LIN {X 0,Y 240.149,Z 360.494,A -85,B 0,C 180,E1 -19958.542,E2 -19958.542} C_VEL
LIN {X 0,Y 236.743,Z 363.17,A -85,B 0,C 180,E1 -19960.941,E2 -19960.941} C_VEL
LIN {X 0,Y 232.958,Z 365.456,A -85,B 0,C 180,E1 -19964.245,E2 -19964.245} C_VEL
LIN {X 0,Y 230.136,Z 366.365,A -85,B 0,C 180,E1 -19967.657,E2 -19967.657} C_VEL
LIN {X 0,Y 228.663,Z 366.29,A -85,B 0,C 180,E1 -19969.595,E2 -19969.595} C_VEL
LIN {X 0,Y 227.257,Z 365.084,A -85,B 0,C 180,E1 -19972.894,E2 -19972.894} C_VEL
LIN {X 0,Y 226.376,Z 362.416,A -85,B 0,C 180,E1 -19976.44,E2 -19976.44} C_VEL
LIN {X 0,Y 225.981,Z 359.392,A -85,B 0,C 180,E1 -19979.109,E2 -19979.109} C_VEL
LIN {X 0,Y 225.959,Z 355.435,A -85,B 0,C 180,E1 -19981.782,E2 -19981.782} C_VEL
LIN {X 0,Y 226.033,Z 350.41,A -85,B 0,C 180,E1 -19984.458,E2 -19984.458} C_VEL
LIN {X 0,Y 226.423,Z 343.052,A -85,B 0,C 180,E1 -19987.58,E2 -19987.58} C_VEL
LIN {X 0,Y 227.138,Z 333.719,A -85,B 0,C 180,E1 -19990.699,E2 -19990.699} C_VEL
LIN {X 0,Y 228.026,Z 323.757,A -85,B 0,C 180,E1 -19993.365,E2 -19993.365} C_VEL
LIN {X 0,Y 229.272,Z 312.636,A -85,B 0,C 180,E1 -19995.786,E2 -19995.786} C_VEL
LIN {X 0,Y 230.346,Z 301.437,A -85,B 0,C 180,E1 -19997.765,E2 -19997.765} C_VEL
LIN {X 0,Y 231.551,Z 289.361,A -85,B 0,C 180,E1 -19999.504,E2 -19999.504} C_VEL
LIN {X 0,Y 231.875,Z 284.182,A -85,B 0,C 180,E1 -20000.139,E2 -20000.139} C_VEL
LIN {X 0,Y 229.783,Z 269.787,A -85,B 0,C 180,E1 -20001.668,E2 -20001.668} C_VEL
LIN {X 0,Y 228.207,Z 255.116,A -85,B 0,C 180,E1 -20002.85,E2 -20002.85} C_VEL
LIN {X 0,Y 228.789,Z 246.393,A -85,B 0,C 180,E1 -20007.437,E2 -20007.437} C_VEL
LIN {X 0,Y 229.412,Z 238.95,A -85,B 0,C 180,E1 -20011.386,E2 -20011.386} C_VEL
LIN {X 0,Y 230.076,Z 231.264,A -85,B 0,C 180,E1 -20015.478,E2 -20015.478} C_VEL
LIN {X 0,Y 229.952,Z 226.244,A -85,B 0,C 180,E1 -20018.23,E2 -20018.23} C_VEL
LIN {X 0,Y 228.576,Z 218.639,A -85,B 0,C 180,E1 -20022.566,E2 -20022.566} C_VEL
LIN {X 0,Y 227.886,Z 215.096,A -85,B 0,C 180,E1 -20024.661,E2 -20024.661} C_VEL
LIN {X 0,Y 227.869,Z 215.294,A -85,B 0,C 180,E1 -20027.269,E2 -20027.269} C_VEL
LIN {X 0,Y 228.539,Z 218.744,A -85,B 0,C 180,E1 -20032.043,E2 -20032.043} C_VEL
LIN {X 0,Y 229.088,Z 222.169,A -85,B 0,C 180,E1 -20036.479,E2 -20036.479} C_VEL
LIN {X 0,Y 229.253,Z 224.421,A -85,B 0,C 180,E1 -20039.135,E2 -20039.135} C_VEL
LIN {X 0,Y 229.175,Z 227.751,A -85,B 0,C 180,E1 -20042.789,E2 -20042.789} C_VEL
LIN {X 0,Y 228.957,Z 231.942,A -85,B 0,C 180,E1 -20047.054,E2 -20047.054} C_VEL
LIN {X 0,Y 232.523,Z 242.538,A -85,B 0,C 180,E1 -20048.242,E2 -20048.242} C_VEL
LIN {X 0,Y 234.853,Z 251.139,A -85,B 0,C 180,E1 -20049.409,E2 -20049.409} C_VEL
LIN {X 0,Y 236.685,Z 260.451,A -85,B 0,C 180,E1 -20050.934,E2 -20050.934} C_VEL
LIN {X 0,Y 237.154,Z 263.439,A -85,B 0,C 180,E1 -20051.499,E2 -20051.499} C_VEL
LIN {X 0,Y 236.153,Z 271.037,A -85,B 0,C 180,E1 -20052.907,E2 -20052.907} C_VEL
LIN {X 0,Y 234.935,Z 277.492,A -85,B 0,C 180,E1 -20054.379,E2 -20054.379} C_VEL
LIN {X 0,Y 233.482,Z 283.544,A -85,B 0,C 180,E1 -20056.064,E2 -20056.064} C_VEL
LIN {X 0,Y 232.2,Z 288.356,A -85,B 0,C 180,E1 -20057.766,E2 -20057.766} C_VEL
LIN {X 0,Y 231.114,Z 292.243,A -85,B 0,C 180,E1 -20059.485,E2 -20059.485} C_VEL
LIN {X 0,Y 230.298,Z 296.589,A -85,B 0,C 180,E1 -20062.105,E2 -20062.105} C_VEL
LIN {X 0,Y 229.216,Z 299.558,A -85,B 0,C 180,E1 -20064.72,E2 -20064.72} C_VEL
LIN {X 0,Y 228.932,Z 300.802,A -85,B 0,C 180,E1 -20066.478,E2 -20066.478} C_VEL
LIN {X 0,Y 228.662,Z 301.565,A -85,B 0,C 180,E1 -20068.236,E2 -20068.236} C_VEL
LIN {X 0,Y 228.557,Z 301.836,A -85,B 0,C 180,E1 -20069.998,E2 -20069.998} C_VEL
LIN {X 0,Y 228.661,Z 301.599,A -85,B 0,C 180,E1 -20071.759,E2 -20071.759} C_VEL
LIN {X 0,Y 228.93,Z 300.884,A -85,B 0,C 180,E1 -20073.518,E2 -20073.518} C_VEL
LIN {X 0,Y 229.213,Z 299.688,A -85,B 0,C 180,E1 -20075.275,E2 -20075.275} C_VEL
LIN {X 0,Y 230.285,Z 296.77,A -85,B 0,C 180,E1 -20077.891,E2 -20077.891} C_VEL
LIN {X 0,Y 231.073,Z 292.516,A -85,B 0,C 180,E1 -20080.512,E2 -20080.512} C_VEL
LIN {X 0,Y 231.808,Z 290.679,A -85,B 0,C 180,E1 -20081.363,E2 -20081.363} C_VEL
LIN {X 0,Y 232.744,Z 286.458,A -85,B 0,C 180,E1 -20083.087,E2 -20083.087} C_VEL
LIN {X 0,Y 234.536,Z 279.688,A -85,B 0,C 180,E1 -20085.198,E2 -20085.198} C_VEL
LIN {X 0,Y 235.91,Z 272.696,A -85,B 0,C 180,E1 -20086.883,E2 -20086.883} C_VEL
LIN {X 0,Y 236.953,Z 265.692,A -85,B 0,C 180,E1 -20088.245,E2 -20088.245} C_VEL
LIN {X 0,Y 237.125,Z 263.241,A -85,B 0,C 180,E1 -20088.68,E2 -20088.68} C_VEL
LIN {X 0,Y 235.737,Z 254.873,A -85,B 0,C 180,E1 -20090.151,E2 -20090.151} C_VEL
LIN {X 0,Y 233.638,Z 246.157,A -85,B 0,C 180,E1 -20091.422,E2 -20091.422} C_VEL
LIN {X 0,Y 230.323,Z 235.832,A -85,B 0,C 180,E1 -20092.688,E2 -20092.688} C_VEL
LIN {X 0,Y 228.951,Z 231.943,A -85,B 0,C 180,E1 -20093.098,E2 -20093.098} C_VEL
LIN {X 0,Y 229.195,Z 227.77,A -85,B 0,C 180,E1 -20097.382,E2 -20097.382} C_VEL
LIN {X 0,Y 229.217,Z 224.148,A -85,B 0,C 180,E1 -20101.412,E2 -20101.412} C_VEL
LIN {X 0,Y 229.06,Z 221.908,A -85,B 0,C 180,E1 -20104.064,E2 -20104.064} C_VEL
LIN {X 0,Y 228.562,Z 218.862,A -85,B 0,C 180,E1 -20107.947,E2 -20107.947} C_VEL
LIN {X 0,Y 227.893,Z 215.434,A -85,B 0,C 180,E1 -20112.72,E2 -20112.72} C_VEL
LIN {X 0,Y 227.863,Z 215.098,A -85,B 0,C 180,E1 -20113.941,E2 -20113.941} C_VEL
LIN {X 0,Y 227.859,Z 215.104,A -85,B 0,C 180,E1 -20117.748,E2 -20117.748} C_VEL
LIN {X 0,Y 227.859,Z 215.097,A -85,B 0,C 180,E1 -20121.912,E2 -20121.912} C_VEL
LIN {X 0,Y 227.877,Z 215.09,A -85,B 0,C 180,E1 -20126.373,E2 -20126.373} C_VEL
LIN {X 0,Y 227.911,Z 215.084,A -85,B 0,C 180,E1 -20130.436,E2 -20130.436} C_VEL
LIN {X 0,Y 227.92,Z 215.082,A -85,B 0,C 180,E1 -20134.425,E2 -20134.425} C_VEL
LIN {X 0,Y 227.953,Z 215.086,A -85,B 0,C 180,E1 -20138.286,E2 -20138.286} C_VEL
LIN {X 0,Y 228.025,Z 215.081,A -85,B 0,C 180,E1 -20142.825,E2 -20142.825} C_VEL
LIN {X 0,Y 228.063,Z 215.078,A -85,B 0,C 180,E1 -20147.543,E2 -20147.543} C_VEL
LIN {X 0,Y 228.257,Z 215.041,A -85,B 0,C 180,E1 -20151.144,E2 -20151.144} C_VEL
LIN {X 0,Y 228.329,Z 215.043,A -85,B 0,C 180,E1 -20152.928,E2 -20152.928} C_VEL
LIN {X 0,Y 228.544,Z 215.014,A -85,B 0,C 180,E1 -20158.238,E2 -20158.238} C_VEL
LIN {X 0,Y 228.543,Z 215.013,A -85,B 0,C 180,E1 -20161.762,E2 -20161.762} C_VEL
LIN {X 0,Y 228.344,Z 215.042,A -85,B 0,C 180,E1 -20167.072,E2 -20167.072} C_VEL
LIN {X 0,Y 228.148,Z 215.062,A -85,B 0,C 180,E1 -20170.651,E2 -20170.651} C_VEL
LIN {X 0,Y 228.031,Z 215.072,A -85,B 0,C 180,E1 -20174.274,E2 -20174.274} C_VEL
LIN {X 0,Y 227.919,Z 215.085,A -85,B 0,C 180,E1 -20177.96,E2 -20177.96} C_VEL
LIN {X 0,Y 227.878,Z 215.101,A -85,B 0,C 180,E1 -20182.304,E2 -20182.304} C_VEL
LIN {X 0,Y 227.893,Z 215.101,A -85,B 0,C 180,E1 -20186.584,E2 -20186.584} C_VEL
LIN {X 0,Y 227.88,Z 215.289,A -85,B 0,C 180,E1 -20188.809,E2 -20188.809} C_VEL
LIN {X 0,Y 229.216,Z 220.372,A -85,B 0,C 180,E1 -20193.497,E2 -20193.497} C_VEL
LIN {X 0,Y 230.426,Z 225.395,A -85,B 0,C 180,E1 -20197.59,E2 -20197.59} C_VEL
LIN {X 0,Y 231.746,Z 231.311,A -85,B 0,C 180,E1 -20201.85,E2 -20201.85} C_VEL
LIN {X 0,Y 233.255,Z 238.212,A -85,B 0,C 180,E1 -20206.313,E2 -20206.313} C_VEL
LIN {X 0,Y 234.535,Z 244.072,A -85,B 0,C 180,E1 -20209.828,E2 -20209.828} C_VEL
LIN {X 0,Y 235.471,Z 248.71,A -85,B 0,C 180,E1 -20212.45,E2 -20212.45} C_VEL
LIN {X 0,Y 235.38,Z 250.389,A -85,B 0,C 180,E1 -20213.311,E2 -20213.311} C_VEL
LIN {X 0,Y 233.997,Z 253.09,A -85,B 0,C 180,E1 -20214.552,E2 -20214.552} C_VEL
LIN {X 0,Y 231.754,Z 255.824,A -85,B 0,C 180,E1 -20215.736,E2 -20215.736} C_VEL
LIN {X 0,Y 227.007,Z 261.454,A -85,B 0,C 180,E1 -20218.199,E2 -20218.199} C_VEL
LIN {X 0,Y 226.091,Z 263.295,A -85,B 0,C 180,E1 -20219.09,E2 -20219.09} C_VEL
LIN {X 0,Y 224.786,Z 267.3,A -85,B 0,C 180,E1 -20221.096,E2 -20221.096} C_VEL
LIN {X 0,Y 225.919,Z 279.544,A -85,B 0,C 180,E1 -20222.011,E2 -20222.011} C_VEL
LIN {X 0,Y 226.392,Z 291.772,A -85,B 0,C 180,E1 -20223.251,E2 -20223.251} C_VEL
LIN {X 0,Y 226.184,Z 302.278,A -85,B 0,C 180,E1 -20224.585,E2 -20224.585} C_VEL
LIN {X 0,Y 225.585,Z 313.26,A -85,B 0,C 180,E1 -20226.355,E2 -20226.355} C_VEL
LIN {X 0,Y 225.14,Z 321.657,A -85,B 0,C 180,E1 -20228.004,E2 -20228.004} C_VEL
LIN {X 0,Y 224.202,Z 327.791,A -85,B 0,C 180,E1 -20229.353,E2 -20229.353} C_VEL
LIN {X 0,Y 222.571,Z 336.194,A -85,B 0,C 180,E1 -20231.596,E2 -20231.596} C_VEL
LIN {X 0,Y 221.338,Z 343.23,A -85,B 0,C 180,E1 -20233.872,E2 -20233.872} C_VEL
LIN {X 0,Y 220.649,Z 348.998,A -85,B 0,C 180,E1 -20236.182,E2 -20236.182} C_VEL
LIN {X 0,Y 220.308,Z 352.862,A -85,B 0,C 180,E1 -20238.035,E2 -20238.035} C_VEL
LIN {X 0,Y 219.852,Z 361.618,A -85,B 0,C 180,E1 -20240.805,E2 -20240.805} C_VEL
LIN {X 0,Y 219.728,Z 369.279,A -85,B 0,C 180,E1 -20243.851,E2 -20243.851} C_VEL
LIN {X 0,Y 219.716,Z 374.223,A -85,B 0,C 180,E1 -20246.334,E2 -20246.334} C_VEL
LIN {X 0,Y 219.799,Z 378.548,A -85,B 0,C 180,E1 -20249.086,E2 -20249.086} C_VEL
LIN {X 0,Y 219.482,Z 381.661,A -85,B 0,C 180,E1 -20251.837,E2 -20251.837} C_VEL
LIN {X 0,Y 218.975,Z 384.309,A -85,B 0,C 180,E1 -20255.528,E2 -20255.528} C_VEL
LIN {X 0,Y 219.193,Z 385.464,A -85,B 0,C 180,E1 -20259.228,E2 -20259.228} C_VEL
LIN {X 0,Y 220.33,Z 385.234,A -85,B 0,C 180,E1 -20262.904,E2 -20262.904} C_VEL
LIN {X 0,Y 222.524,Z 383.673,A -85,B 0,C 180,E1 -20266.516,E2 -20266.516} C_VEL
LIN {X 0,Y 225.922,Z 380.789,A -85,B 0,C 180,E1 -20270.012,E2 -20270.012} C_VEL
LIN {X 0,Y 230.072,Z 376.537,A -85,B 0,C 180,E1 -20273.4,E2 -20273.4} C_VEL
LIN {X 0,Y 234.016,Z 372.441,A -85,B 0,C 180,E1 -20275.817,E2 -20275.817} C_VEL
LIN {X 0,Y 240.311,Z 365.58,A -85,B 0,C 180,E1 -20278.854,E2 -20278.854} C_VEL
LIN {X 0,Y 246.571,Z 358.222,A -85,B 0,C 180,E1 -20281.346,E2 -20281.346} C_VEL
LIN {X 0,Y 253.528,Z 349.34,A -85,B 0,C 180,E1 -20283.673,E2 -20283.673} C_VEL
LIN {X 0,Y 259.702,Z 340.339,A -85,B 0,C 180,E1 -20285.677,E2 -20285.677} C_VEL
LIN {X 0,Y 264.058,Z 332.941,A -85,B 0,C 180,E1 -20287.267,E2 -20287.267} C_VEL
LIN {X 0,Y 268.671,Z 323.71,A -85,B 0,C 180,E1 -20289.382,E2 -20289.382} C_VEL
LIN {X 0,Y 271.657,Z 316.985,A -85,B 0,C 180,E1 -20291.061,E2 -20291.061} C_VEL
LIN {X 0,Y 272.448,Z 315.16,A -85,B 0,C 180,E1 -20291.576,E2 -20291.576} C_VEL
LIN {X 0,Y 271.791,Z 313.866,A -85,B 0,C 180,E1 -20293.612,E2 -20293.612} C_VEL
LIN {X 0,Y 271.036,Z 313.826,A -85,B 0,C 180,E1 -20295.564,E2 -20295.564} C_VEL
LIN {X 0,Y 270.322,Z 314.74,A -85,B 0,C 180,E1 -20297.471,E2 -20297.471} C_VEL
LIN {X 0,Y 269.382,Z 316.745,A -85,B 0,C 180,E1 -20299.29,E2 -20299.29} C_VEL
LIN {X 0,Y 267.011,Z 322.182,A -85,B 0,C 180,E1 -20302.154,E2 -20302.154} C_VEL
LIN {X 0,Y 265.102,Z 326.951,A -85,B 0,C 180,E1 -20304.322,E2 -20304.322} C_VEL
LIN {X 0,Y 263.807,Z 329.919,A -85,B 0,C 180,E1 -20305.52,E2 -20305.52} C_VEL
LIN {X 0,Y 255.753,Z 340.457,A -85,B 0,C 180,E1 -20308.063,E2 -20308.063} C_VEL
LIN {X 0,Y 249.21,Z 347.925,A -85,B 0,C 180,E1 -20310.428,E2 -20310.428} C_VEL
LIN {X 0,Y 242.343,Z 354.828,A -85,B 0,C 180,E1 -20313.288,E2 -20313.288} C_VEL
LIN {X 0,Y 236.377,Z 360.018,A -85,B 0,C 180,E1 -20316.335,E2 -20316.335} C_VEL
LIN {X 0,Y 232.456,Z 362.935,A -85,B 0,C 180,E1 -20318.727,E2 -20318.727} C_VEL
LIN {X 0,Y 228.124,Z 365.563,A -85,B 0,C 180,E1 -20322.057,E2 -20322.057} C_VEL
LIN {X 0,Y 224.573,Z 366.846,A -85,B 0,C 180,E1 -20325.501,E2 -20325.501} C_VEL
LIN {X 0,Y 223.238,Z 366.942,A -85,B 0,C 180,E1 -20327.269,E2 -20327.269} C_VEL
LIN {X 0,Y 221.465,Z 366.566,A -85,B 0,C 180,E1 -20329.669,E2 -20329.669} C_VEL
LIN {X 0,Y 220.21,Z 365.192,A -85,B 0,C 180,E1 -20332.666,E2 -20332.666} C_VEL
LIN {X 0,Y 219.718,Z 363.902,A -85,B 0,C 180,E1 -20334.494,E2 -20334.494} C_VEL
LIN {X 0,Y 219.017,Z 360.148,A -85,B 0,C 180,E1 -20338.161,E2 -20338.161} C_VEL
LIN {X 0,Y 218.852,Z 356.283,A -85,B 0,C 180,E1 -20340.92,E2 -20340.92} C_VEL
LIN {X 0,Y 218.96,Z 351.387,A -85,B 0,C 180,E1 -20343.681,E2 -20343.681} C_VEL
LIN {X 0,Y 219.208,Z 344.201,A -85,B 0,C 180,E1 -20346.905,E2 -20346.905} C_VEL
LIN {X 0,Y 219.775,Z 336.514,A -85,B 0,C 180,E1 -20349.665,E2 -20349.665} C_VEL
LIN {X 0,Y 220.62,Z 327.16,A -85,B 0,C 180,E1 -20352.417,E2 -20352.417} C_VEL
LIN {X 0,Y 221.671,Z 316.694,A -85,B 0,C 180,E1 -20354.928,E2 -20354.928} C_VEL
LIN {X 0,Y 222.9,Z 305.135,A -85,B 0,C 180,E1 -20357.193,E2 -20357.193} C_VEL
LIN {X 0,Y 223.982,Z 293.762,A -85,B 0,C 180,E1 -20358.999,E2 -20358.999} C_VEL
LIN {X 0,Y 224.733,Z 284.257,A -85,B 0,C 180,E1 -20360.247,E2 -20360.247} C_VEL
LIN {X 0,Y 222.818,Z 271.045,A -85,B 0,C 180,E1 -20361.705,E2 -20361.705} C_VEL
LIN {X 0,Y 221.224,Z 257.082,A -85,B 0,C 180,E1 -20362.88,E2 -20362.88} C_VEL
LIN {X 0,Y 221.161,Z 255.442,A -85,B 0,C 180,E1 -20363.034,E2 -20363.034} C_VEL
LIN {X 0,Y 221.732,Z 247.231,A -85,B 0,C 180,E1 -20367.437,E2 -20367.437} C_VEL
LIN {X 0,Y 222.518,Z 237.916,A -85,B 0,C 180,E1 -20372.475,E2 -20372.475} C_VEL
LIN {X 0,Y 223.08,Z 231.879,A -85,B 0,C 180,E1 -20375.753,E2 -20375.753} C_VEL
LIN {X 0,Y 223,Z 227.838,A -85,B 0,C 180,E1 -20378.008,E2 -20378.008} C_VEL
LIN {X 0,Y 221.917,Z 221.47,A -85,B 0,C 180,E1 -20381.687,E2 -20381.687} C_VEL
LIN {X 0,Y 220.848,Z 215.972,A -85,B 0,C 180,E1 -20384.962,E2 -20384.962} C_VEL
LIN {X 0,Y 220.859,Z 216.006,A -85,B 0,C 180,E1 -20385.565,E2 -20385.565} C_VEL
LIN {X 0,Y 221.464,Z 219.399,A -85,B 0,C 180,E1 -20390.601,E2 -20390.601} C_VEL
LIN {X 0,Y 221.819,Z 221.151,A -85,B 0,C 180,E1 -20392.985,E2 -20392.985} C_VEL
LIN {X 0,Y 222.062,Z 222.974,A -85,B 0,C 180,E1 -20395.374,E2 -20395.374} C_VEL
LIN {X 0,Y 222.33,Z 226.478,A -85,B 0,C 180,E1 -20399.615,E2 -20399.615} C_VEL
LIN {X 0,Y 222.177,Z 230.205,A -85,B 0,C 180,E1 -20403.712,E2 -20403.712} C_VEL
LIN {X 0,Y 222.019,Z 232.583,A -85,B 0,C 180,E1 -20406.171,E2 -20406.171} C_VEL
LIN {X 0,Y 225.819,Z 243.551,A -85,B 0,C 180,E1 -20407.497,E2 -20407.497} C_VEL
LIN {X 0,Y 228.213,Z 252.528,A -85,B 0,C 180,E1 -20408.781,E2 -20408.781} C_VEL
LIN {X 0,Y 229.971,Z 261.716,A -85,B 0,C 180,E1 -20410.355,E2 -20410.355} C_VEL
LIN {X 0,Y 230.456,Z 264.797,A -85,B 0,C 180,E1 -20410.976,E2 -20410.976} C_VEL
LIN {X 0,Y 229.462,Z 272.136,A -85,B 0,C 180,E1 -20412.393,E2 -20412.393} C_VEL
LIN {X 0,Y 228.187,Z 278.548,A -85,B 0,C 180,E1 -20413.905,E2 -20413.905} C_VEL
LIN {X 0,Y 226.674,Z 284.563,A -85,B 0,C 180,E1 -20415.636,E2 -20415.636} C_VEL
LIN {X 0,Y 225.336,Z 289.356,A -85,B 0,C 180,E1 -20417.387,E2 -20417.387} C_VEL
LIN {X 0,Y 224.205,Z 293.231,A -85,B 0,C 180,E1 -20419.157,E2 -20419.157} C_VEL
LIN {X 0,Y 223.338,Z 297.567,A -85,B 0,C 180,E1 -20421.857,E2 -20421.857} C_VEL
LIN {X 0,Y 222.219,Z 300.534,A -85,B 0,C 180,E1 -20424.553,E2 -20424.553} C_VEL
LIN {X 0,Y 221.918,Z 301.776,A -85,B 0,C 180,E1 -20426.366,E2 -20426.366} C_VEL
LIN {X 0,Y 221.638,Z 302.538,A -85,B 0,C 180,E1 -20428.181,E2 -20428.181} C_VEL
LIN {X 0,Y 221.529,Z 302.81,A -85,B 0,C 180,E1 -20429.998,E2 -20429.998} C_VEL
LIN {X 0,Y 221.636,Z 302.573,A -85,B 0,C 180,E1 -20431.815,E2 -20431.815} C_VEL
LIN {X 0,Y 221.916,Z 301.858,A -85,B 0,C 180,E1 -20433.629,E2 -20433.629} C_VEL
LIN {X 0,Y 222.217,Z 300.662,A -85,B 0,C 180,E1 -20435.442,E2 -20435.442} C_VEL
LIN {X 0,Y 223.326,Z 297.746,A -85,B 0,C 180,E1 -20438.139,E2 -20438.139} C_VEL
LIN {X 0,Y 224.164,Z 293.502,A -85,B 0,C 180,E1 -20440.84,E2 -20440.84} C_VEL
LIN {X 0,Y 224.92,Z 291.671,A -85,B 0,C 180,E1 -20441.716,E2 -20441.716} C_VEL
LIN {X 0,Y 225.906,Z 287.465,A -85,B 0,C 180,E1 -20443.491,E2 -20443.491} C_VEL
LIN {X 0,Y 227.771,Z 280.73,A -85,B 0,C 180,E1 -20445.661,E2 -20445.661} C_VEL
LIN {X 0,Y 229.209,Z 273.788,A -85,B 0,C 180,E1 -20447.392,E2 -20447.392} C_VEL
LIN {X 0,Y 230.261,Z 267.189,A -85,B 0,C 180,E1 -20448.73,E2 -20448.73} C_VEL
LIN {X 0,Y 230.424,Z 264.33,A -85,B 0,C 180,E1 -20449.259,E2 -20449.259} C_VEL
LIN {X 0,Y 229.076,Z 256.108,A -85,B 0,C 180,E1 -20450.773,E2 -20450.773} C_VEL
LIN {X 0,Y 226.772,Z 246.713,A -85,B 0,C 180,E1 -20452.213,E2 -20452.213} C_VEL
LIN {X 0,Y 223.456,Z 236.681,A -85,B 0,C 180,E1 -20453.512,E2 -20453.512} C_VEL
LIN {X 0,Y 222.037,Z 232.592,A -85,B 0,C 180,E1 -20453.991,E2 -20453.991} C_VEL
LIN {X 0,Y 222.273,Z 228.51,A -85,B 0,C 180,E1 -20458.31,E2 -20458.31} C_VEL
LIN {X 0,Y 222.316,Z 225.809,A -85,B 0,C 180,E1 -20461.4,E2 -20461.4} C_VEL
LIN {X 0,Y 222.084,Z 223.068,A -85,B 0,C 180,E1 -20464.721,E2 -20464.721} C_VEL
LIN {X 0,Y 221.76,Z 220.89,A -85,B 0,C 180,E1 -20467.599,E2 -20467.599} C_VEL
LIN {X 0,Y 221.136,Z 217.866,A -85,B 0,C 180,E1 -20471.864,E2 -20471.864} C_VEL
LIN {X 0,Y 220.794,Z 215.983,A -85,B 0,C 180,E1 -20474.99,E2 -20474.99} C_VEL
LIN {X 0,Y 220.797,Z 215.976,A -85,B 0,C 180,E1 -20479.807,E2 -20479.807} C_VEL
LIN {X 0,Y 220.817,Z 215.971,A -85,B 0,C 180,E1 -20482.791,E2 -20482.791} C_VEL
LIN {X 0,Y 220.813,Z 215.973,A -85,B 0,C 180,E1 -20487.243,E2 -20487.243} C_VEL
LIN {X 0,Y 220.829,Z 215.97,A -85,B 0,C 180,E1 -20491.485,E2 -20491.485} C_VEL
LIN {X 0,Y 220.858,Z 215.961,A -85,B 0,C 180,E1 -20495.564,E2 -20495.564} C_VEL
LIN {X 0,Y 220.883,Z 215.957,A -85,B 0,C 180,E1 -20499.513,E2 -20499.513} C_VEL
LIN {X 0,Y 221.007,Z 215.948,A -85,B 0,C 180,E1 -20503.369,E2 -20503.369} C_VEL
LIN {X 0,Y 221.002,Z 215.956,A -85,B 0,C 180,E1 -20507.138,E2 -20507.138} C_VEL
LIN {X 0,Y 221.195,Z 215.918,A -85,B 0,C 180,E1 -20510.859,E2 -20510.859} C_VEL
LIN {X 0,Y 221.261,Z 215.923,A -85,B 0,C 180,E1 -20512.701,E2 -20512.701} C_VEL
LIN {X 0,Y 221.502,Z 215.891,A -85,B 0,C 180,E1 -20518.182,E2 -20518.182} C_VEL
LIN {X 0,Y 221.501,Z 215.89,A -85,B 0,C 180,E1 -20521.818,E2 -20521.818} C_VEL
LIN {X 0,Y 221.295,Z 215.92,A -85,B 0,C 180,E1 -20527.298,E2 -20527.298} C_VEL
LIN {X 0,Y 221.095,Z 215.944,A -85,B 0,C 180,E1 -20530.995,E2 -20530.995} C_VEL
LIN {X 0,Y 220.967,Z 215.954,A -85,B 0,C 180,E1 -20536.634,E2 -20536.634} C_VEL
LIN {X 0,Y 220.841,Z 215.977,A -85,B 0,C 180,E1 -20540.491,E2 -20540.491} C_VEL
LIN {X 0,Y 220.787,Z 215.984,A -85,B 0,C 180,E1 -20544.444,E2 -20544.444} C_VEL
LIN {X 0,Y 220.842,Z 216.176,A -85,B 0,C 180,E1 -20546.999,E2 -20546.999} C_VEL
LIN {X 0,Y 221.903,Z 220.35,A -85,B 0,C 180,E1 -20551.231,E2 -20551.231} C_VEL
LIN {X 0,Y 223.162,Z 225.299,A -85,B 0,C 180,E1 -20555.634,E2 -20555.634} C_VEL
LIN {X 0,Y 224.438,Z 230.91,A -85,B 0,C 180,E1 -20559.936,E2 -20559.936} C_VEL
LIN {X 0,Y 225.73,Z 237.039,A -85,B 0,C 180,E1 -20564.271,E2 -20564.271} C_VEL
LIN {X 0,Y 227.335,Z 244.142,A -85,B 0,C 180,E1 -20568.773,E2 -20568.773} C_VEL
LIN {X 0,Y 228.798,Z 251.307,A -85,B 0,C 180,E1 -20573.001,E2 -20573.001} C_VEL
LIN {X 0,Y 229.26,Z 253.766,A -85,B 0,C 180,E1 -20574.38,E2 -20574.38} C_VEL
LIN {X 0,Y 228.891,Z 255.747,A -85,B 0,C 180,E1 -20575.391,E2 -20575.391} C_VEL
LIN {X 0,Y 226.091,Z 263.295,A -85,B 0,C 180,E1 -20579.09,E2 -20579.09} C_VEL
LIN {X 0,Y 225.363,Z 265.52,A -85,B 0,C 180,E1 -20579.858,E2 -20579.858} C_VEL
LIN {X 0,Y 224.186,Z 269.261,A -85,B 0,C 180,E1 -20580.582,E2 -20580.582} C_VEL
LIN {X 0,Y 222.403,Z 275.408,A -85,B 0,C 180,E1 -20581.255,E2 -20581.255} C_VEL
LIN {X 0,Y 220.569,Z 284.065,A -85,B 0,C 180,E1 -20581.808,E2 -20581.808} C_VEL
LIN {X 0,Y 219.821,Z 289.449,A -85,B 0,C 180,E1 -20582.291,E2 -20582.291} C_VEL
LIN {X 0,Y 219.753,Z 291.207,A -85,B 0,C 180,E1 -20582.487,E2 -20582.487} C_VEL
LIN {X 0,Y 219.552,Z 300.931,A -85,B 0,C 180,E1 -20583.76,E2 -20583.76} C_VEL
LIN {X 0,Y 218.927,Z 310.79,A -85,B 0,C 180,E1 -20585.337,E2 -20585.337} C_VEL
LIN {X 0,Y 218.329,Z 320.512,A -85,B 0,C 180,E1 -20587.28,E2 -20587.28} C_VEL
LIN {X 0,Y 217.498,Z 326.71,A -85,B 0,C 180,E1 -20588.686,E2 -20588.686} C_VEL
LIN {X 0,Y 215.767,Z 335.145,A -85,B 0,C 180,E1 -20590.993,E2 -20590.993} C_VEL
LIN {X 0,Y 214.448,Z 342.196,A -85,B 0,C 180,E1 -20593.339,E2 -20593.339} C_VEL
LIN {X 0,Y 213.679,Z 347.978,A -85,B 0,C 180,E1 -20595.722,E2 -20595.722} C_VEL
LIN {X 0,Y 213.19,Z 353.878,A -85,B 0,C 180,E1 -20598.715,E2 -20598.715} C_VEL
LIN {X 0,Y 212.874,Z 361.965,A -85,B 0,C 180,E1 -20601.46,E2 -20601.46} C_VEL
LIN {X 0,Y 212.751,Z 368.792,A -85,B 0,C 180,E1 -20604.315,E2 -20604.315} C_VEL
LIN {X 0,Y 212.777,Z 374.195,A -85,B 0,C 180,E1 -20607.163,E2 -20607.163} C_VEL
LIN {X 0,Y 212.78,Z 378.34,A -85,B 0,C 180,E1 -20610.002,E2 -20610.002} C_VEL
LIN {X 0,Y 212.48,Z 380.44,A -85,B 0,C 180,E1 -20611.898,E2 -20611.898} C_VEL
LIN {X 0,Y 211.955,Z 383.4,A -85,B 0,C 180,E1 -20615.877,E2 -20615.877} C_VEL
LIN {X 0,Y 212.198,Z 384.747,A -85,B 0,C 180,E1 -20619.534,E2 -20619.534} C_VEL
LIN {X 0,Y 213.377,Z 384.841,A -85,B 0,C 180,E1 -20623.332,E2 -20623.332} C_VEL
LIN {X 0,Y 215.722,Z 383.594,A -85,B 0,C 180,E1 -20627.053,E2 -20627.053} C_VEL
LIN {X 0,Y 219.253,Z 381.038,A -85,B 0,C 180,E1 -20630.649,E2 -20630.649} C_VEL
LIN {X 0,Y 223.618,Z 377.201,A -85,B 0,C 180,E1 -20634.117,E2 -20634.117} C_VEL
LIN {X 0,Y 227.712,Z 373.426,A -85,B 0,C 180,E1 -20636.587,E2 -20636.587} C_VEL
LIN {X 0,Y 234.245,Z 367.102,A -85,B 0,C 180,E1 -20639.675,E2 -20639.675} C_VEL
LIN {X 0,Y 241.705,Z 359.138,A -85,B 0,C 180,E1 -20642.545,E2 -20642.545} C_VEL
LIN {X 0,Y 249.994,Z 349.388,A -85,B 0,C 180,E1 -20645.194,E2 -20645.194} C_VEL
LIN {X 0,Y 257.287,Z 339.395,A -85,B 0,C 180,E1 -20647.48,E2 -20647.48} C_VEL
LIN {X 0,Y 262.528,Z 330.812,A -85,B 0,C 180,E1 -20649.481,E2 -20649.481} C_VEL
LIN {X 0,Y 267.124,Z 322.347,A -85,B 0,C 180,E1 -20651.624,E2 -20651.624} C_VEL
LIN {X 0,Y 267.523,Z 321.562,A -85,B 0,C 180,E1 -20651.836,E2 -20651.836} C_VEL
LIN {X 0,Y 267.903,Z 320.091,A -85,B 0,C 180,E1 -20652.732,E2 -20652.732} C_VEL
LIN {X 0,Y 266.968,Z 319.57,A -85,B 0,C 180,E1 -20655.301,E2 -20655.301} C_VEL
LIN {X 0,Y 266.366,Z 320.061,A -85,B 0,C 180,E1 -20656.685,E2 -20656.685} C_VEL
LIN {X 0,Y 265.324,Z 321.668,A -85,B 0,C 180,E1 -20658.531,E2 -20658.531} C_VEL
LIN {X 0,Y 263.273,Z 325.288,A -85,B 0,C 180,E1 -20660.73,E2 -20660.73} C_VEL
LIN {X 0,Y 260.381,Z 330.97,A -85,B 0,C 180,E1 -20663.572,E2 -20663.572} C_VEL
LIN {X 0,Y 259.448,Z 332.693,A -85,B 0,C 180,E1 -20664.358,E2 -20664.358} C_VEL
LIN {X 0,Y 258.699,Z 333.847,A -85,B 0,C 180,E1 -20664.728,E2 -20664.728} C_VEL
LIN {X 0,Y 251.204,Z 342.622,A -85,B 0,C 180,E1 -20666.937,E2 -20666.937} C_VEL
LIN {X 0,Y 243.42,Z 350.677,A -85,B 0,C 180,E1 -20669.652,E2 -20669.652} C_VEL
LIN {X 0,Y 236.291,Z 357.009,A -85,B 0,C 180,E1 -20672.547,E2 -20672.547} C_VEL
LIN {X 0,Y 231.534,Z 360.704,A -85,B 0,C 180,E1 -20674.852,E2 -20674.852} C_VEL
LIN {X 0,Y 226.005,Z 364.371,A -85,B 0,C 180,E1 -20678.089,E2 -20678.089} C_VEL
LIN {X 0,Y 221.465,Z 366.594,A -85,B 0,C 180,E1 -20681.498,E2 -20681.498} C_VEL
LIN {X 0,Y 217.758,Z 367.503,A -85,B 0,C 180,E1 -20685.037,E2 -20685.037} C_VEL
LIN {X 0,Y 216.353,Z 367.451,A -85,B 0,C 180,E1 -20686.857,E2 -20686.857} C_VEL
LIN {X 0,Y 214.219,Z 366.637,A -85,B 0,C 180,E1 -20689.82,E2 -20689.82} C_VEL
LIN {X 0,Y 213.17,Z 365.2,A -85,B 0,C 180,E1 -20692.422,E2 -20692.422} C_VEL
LIN {X 0,Y 212.264,Z 361.928,A -85,B 0,C 180,E1 -20696.203,E2 -20696.203} C_VEL
LIN {X 0,Y 211.843,Z 358.448,A -85,B 0,C 180,E1 -20699.05,E2 -20699.05} C_VEL
LIN {X 0,Y 211.832,Z 354.006,A -85,B 0,C 180,E1 -20701.901,E2 -20701.901} C_VEL
LIN {X 0,Y 211.94,Z 347.942,A -85,B 0,C 180,E1 -20705.006,E2 -20705.006} C_VEL
LIN {X 0,Y 212.367,Z 340.417,A -85,B 0,C 180,E1 -20708.085,E2 -20708.085} C_VEL
LIN {X 0,Y 213.086,Z 331.873,A -85,B 0,C 180,E1 -20710.932,E2 -20710.932} C_VEL
LIN {X 0,Y 213.842,Z 323.302,A -85,B 0,C 180,E1 -20713.301,E2 -20713.301} C_VEL
LIN {X 0,Y 215.114,Z 311.996,A -85,B 0,C 180,E1 -20715.88,E2 -20715.88} C_VEL
LIN {X 0,Y 216.226,Z 300.655,A -85,B 0,C 180,E1 -20717.986,E2 -20717.986} C_VEL
LIN {X 0,Y 217.534,Z 287.556,A -85,B 0,C 180,E1 -20719.926,E2 -20719.926} C_VEL
LIN {X 0,Y 217.48,Z 283.742,A -85,B 0,C 180,E1 -20720.416,E2 -20720.416} C_VEL
LIN {X 0,Y 215.612,Z 270.687,A -85,B 0,C 180,E1 -20721.889,E2 -20721.889} C_VEL
LIN {X 0,Y 214.101,Z 255.79,A -85,B 0,C 180,E1 -20723.198,E2 -20723.198} C_VEL
LIN {X 0,Y 214.728,Z 247.192,A -85,B 0,C 180,E1 -20727.903,E2 -20727.903} C_VEL
LIN {X 0,Y 215.5,Z 238.479,A -85,B 0,C 180,E1 -20732.708,E2 -20732.708} C_VEL
LIN {X 0,Y 216.081,Z 231.82,A -85,B 0,C 180,E1 -20736.412,E2 -20736.412} C_VEL
LIN {X 0,Y 215.856,Z 227.993,A -85,B 0,C 180,E1 -20738.607,E2 -20738.607} C_VEL
LIN {X 0,Y 214.663,Z 221.38,A -85,B 0,C 180,E1 -20742.509,E2 -20742.509} C_VEL
LIN {X 0,Y 213.907,Z 217.488,A -85,B 0,C 180,E1 -20744.911,E2 -20744.911} C_VEL
LIN {X 0,Y 214.371,Z 220.165,A -85,B 0,C 180,E1 -20749.026,E2 -20749.026} C_VEL
LIN {X 0,Y 214.736,Z 222.052,A -85,B 0,C 180,E1 -20751.766,E2 -20751.766} C_VEL
LIN {X 0,Y 215.096,Z 224.258,A -85,B 0,C 180,E1 -20754.77,E2 -20754.77} C_VEL
LIN {X 0,Y 215.417,Z 227.208,A -85,B 0,C 180,E1 -20758.531,E2 -20758.531} C_VEL
LIN {X 0,Y 215.304,Z 230.953,A -85,B 0,C 180,E1 -20762.804,E2 -20762.804} C_VEL
LIN {X 0,Y 215.106,Z 233.264,A -85,B 0,C 180,E1 -20765.26,E2 -20765.26} C_VEL
LIN {X 0,Y 219.154,Z 244.783,A -85,B 0,C 180,E1 -20766.728,E2 -20766.728} C_VEL
LIN {X 0,Y 221.588,Z 253.883,A -85,B 0,C 180,E1 -20768.112,E2 -20768.112} C_VEL
LIN {X 0,Y 223.308,Z 262.958,A -85,B 0,C 180,E1 -20769.743,E2 -20769.743} C_VEL
LIN {X 0,Y 223.782,Z 266.142,A -85,B 0,C 180,E1 -20770.42,E2 -20770.42} C_VEL
LIN {X 0,Y 222.983,Z 272.221,A -85,B 0,C 180,E1 -20771.626,E2 -20771.626} C_VEL
LIN {X 0,Y 221.823,Z 277.934,A -85,B 0,C 180,E1 -20772.956,E2 -20772.956} C_VEL
LIN {X 0,Y 220.245,Z 284.243,A -85,B 0,C 180,E1 -20774.734,E2 -20774.734} C_VEL
LIN {X 0,Y 218.483,Z 290.358,A -85,B 0,C 180,E1 -20776.985,E2 -20776.985} C_VEL
LIN {X 0,Y 217.305,Z 294.22,A -85,B 0,C 180,E1 -20778.808,E2 -20778.808} C_VEL
LIN {X 0,Y 216.383,Z 298.544,A -85,B 0,C 180,E1 -20781.593,E2 -20781.593} C_VEL
LIN {X 0,Y 215.225,Z 301.511,A -85,B 0,C 180,E1 -20784.376,E2 -20784.376} C_VEL
LIN {X 0,Y 214.905,Z 302.751,A -85,B 0,C 180,E1 -20786.247,E2 -20786.247} C_VEL
LIN {X 0,Y 214.614,Z 303.512,A -85,B 0,C 180,E1 -20788.121,E2 -20788.121} C_VEL
LIN {X 0,Y 214.502,Z 303.784,A -85,B 0,C 180,E1 -20789.998,E2 -20789.998} C_VEL
LIN {X 0,Y 214.613,Z 303.546,A -85,B 0,C 180,E1 -20791.874,E2 -20791.874} C_VEL
LIN {X 0,Y 214.903,Z 302.832,A -85,B 0,C 180,E1 -20793.748,E2 -20793.748} C_VEL
LIN {X 0,Y 215.222,Z 301.637,A -85,B 0,C 180,E1 -20795.619,E2 -20795.619} C_VEL
LIN {X 0,Y 216.37,Z 298.721,A -85,B 0,C 180,E1 -20798.402,E2 -20798.402} C_VEL
LIN {X 0,Y 217.263,Z 294.488,A -85,B 0,C 180,E1 -20801.189,E2 -20801.189} C_VEL
LIN {X 0,Y 218.041,Z 292.662,A -85,B 0,C 180,E1 -20802.091,E2 -20802.091} C_VEL
LIN {X 0,Y 219.08,Z 288.47,A -85,B 0,C 180,E1 -20803.919,E2 -20803.919} C_VEL
LIN {X 0,Y 221.022,Z 281.769,A -85,B 0,C 180,E1 -20806.152,E2 -20806.152} C_VEL
LIN {X 0,Y 222.715,Z 273.866,A -85,B 0,C 180,E1 -20808.154,E2 -20808.154} C_VEL
LIN {X 0,Y 223.864,Z 266.524,A -85,B 0,C 180,E1 -20809.639,E2 -20809.639} C_VEL
LIN {X 0,Y 222.742,Z 259.099,A -85,B 0,C 180,E1 -20811.122,E2 -20811.122} C_VEL
LIN {X 0,Y 220.775,Z 250.236,A -85,B 0,C 180,E1 -20812.606,E2 -20812.606} C_VEL
LIN {X 0,Y 217.663,Z 240.243,A -85,B 0,C 180,E1 -20814.032,E2 -20814.032} C_VEL
LIN {X 0,Y 215.126,Z 233.247,A -85,B 0,C 180,E1 -20814.93,E2 -20814.93} C_VEL
LIN {X 0,Y 215.353,Z 230.229,A -85,B 0,C 180,E1 -20818.219,E2 -20818.219} C_VEL
LIN {X 0,Y 215.367,Z 227.001,A -85,B 0,C 180,E1 -20821.956,E2 -20821.956} C_VEL
LIN {X 0,Y 215.017,Z 223.798,A -85,B 0,C 180,E1 -20826.036,E2 -20826.036} C_VEL
LIN {X 0,Y 214.766,Z 222.091,A -85,B 0,C 180,E1 -20828.441,E2 -20828.441} C_VEL
LIN {X 0,Y 214.076,Z 218.486,A -85,B 0,C 180,E1 -20833.759,E2 -20833.759} C_VEL
LIN {X 0,Y 213.751,Z 216.854,A -85,B 0,C 180,E1 -20836.657,E2 -20836.657} C_VEL
LIN {X 0,Y 213.73,Z 216.861,A -85,B 0,C 180,E1 -20841.334,E2 -20841.334} C_VEL
LIN {X 0,Y 213.755,Z 216.849,A -85,B 0,C 180,E1 -20846.017,E2 -20846.017} C_VEL
LIN {X 0,Y 213.773,Z 216.845,A -85,B 0,C 180,E1 -20850.453,E2 -20850.453} C_VEL
LIN {X 0,Y 213.792,Z 216.84,A -85,B 0,C 180,E1 -20854.7,E2 -20854.7} C_VEL
LIN {X 0,Y 213.81,Z 216.841,A -85,B 0,C 180,E1 -20858.803,E2 -20858.803} C_VEL
LIN {X 0,Y 213.934,Z 216.836,A -85,B 0,C 180,E1 -20862.803,E2 -20862.803} C_VEL
LIN {X 0,Y 213.943,Z 216.832,A -85,B 0,C 180,E1 -20866.706,E2 -20866.706} C_VEL
LIN {X 0,Y 214.132,Z 216.795,A -85,B 0,C 180,E1 -20870.555,E2 -20870.555} C_VEL
LIN {X 0,Y 214.198,Z 216.802,A -85,B 0,C 180,E1 -20872.458,E2 -20872.458} C_VEL
LIN {X 0,Y 214.435,Z 216.772,A -85,B 0,C 180,E1 -20878.122,E2 -20878.122} C_VEL
LIN {X 0,Y 214.54,Z 216.744,A -85,B 0,C 180,E1 -20880,E2 -20880} C_VEL
LIN {X 0,Y 214.434,Z 216.771,A -85,B 0,C 180,E1 -20881.878,E2 -20881.878} C_VEL
LIN {X 0,Y 214.23,Z 216.799,A -85,B 0,C 180,E1 -20887.54,E2 -20887.54} C_VEL
LIN {X 0,Y 214.01,Z 216.828,A -85,B 0,C 180,E1 -20891.364,E2 -20891.364} C_VEL
LIN {X 0,Y 213.894,Z 216.842,A -85,B 0,C 180,E1 -20895.24,E2 -20895.24} C_VEL
LIN {X 0,Y 213.785,Z 216.856,A -85,B 0,C 180,E1 -20899.192,E2 -20899.192} C_VEL
LIN {X 0,Y 213.773,Z 216.86,A -85,B 0,C 180,E1 -20903.236,E2 -20903.236} C_VEL
LIN {X 0,Y 213.757,Z 216.874,A -85,B 0,C 180,E1 -20904.784,E2 -20904.784} C_VEL
LIN {X 0,Y 214.775,Z 220.988,A -85,B 0,C 180,E1 -20909.396,E2 -20909.396} C_VEL
LIN {X 0,Y 215.915,Z 225.374,A -85,B 0,C 180,E1 -20913.597,E2 -20913.597} C_VEL
LIN {X 0,Y 217.102,Z 230.531,A -85,B 0,C 180,E1 -20917.957,E2 -20917.957} C_VEL
LIN {X 0,Y 218.442,Z 236.62,A -85,B 0,C 180,E1 -20922.504,E2 -20922.504} C_VEL
LIN {X 0,Y 219.971,Z 243.631,A -85,B 0,C 180,E1 -20927.294,E2 -20927.294} C_VEL
LIN {X 0,Y 221.373,Z 250.547,A -85,B 0,C 180,E1 -20931.599,E2 -20931.599} C_VEL
LIN {X 0,Y 222.266,Z 254.965,A -85,B 0,C 180,E1 -20934.203,E2 -20934.203} C_VEL
LIN {X 0,Y 221.519,Z 257.586,A -85,B 0,C 180,E1 -20935.577,E2 -20935.577} C_VEL
LIN {X 0,Y 218.176,Z 266.82,A -85,B 0,C 180,E1 -20940.244,E2 -20940.244} C_VEL
LIN {X 0,Y 219.285,Z 278.731,A -85,B 0,C 180,E1 -20941.174,E2 -20941.174} C_VEL
LIN {X 0,Y 219.753,Z 291.207,A -85,B 0,C 180,E1 -20942.487,E2 -20942.487} C_VEL
LIN {X 0,Y 219.061,Z 294.878,A -85,B 0,C 180,E1 -20942.856,E2 -20942.856} C_VEL
LIN {X 0,Y 216.136,Z 300.693,A -85,B 0,C 180,E1 -20943.354,E2 -20943.354} C_VEL
LIN {X 0,Y 213.093,Z 306.288,A -85,B 0,C 180,E1 -20943.967,E2 -20943.967} C_VEL
LIN {X 0,Y 212.231,Z 309.612,A -85,B 0,C 180,E1 -20944.514,E2 -20944.514} C_VEL
LIN {X 0,Y 211.565,Z 319.369,A -85,B 0,C 180,E1 -20946.51,E2 -20946.51} C_VEL
LIN {X 0,Y 210.848,Z 325.627,A -85,B 0,C 180,E1 -20947.979,E2 -20947.979} C_VEL
LIN {X 0,Y 209.019,Z 334.102,A -85,B 0,C 180,E1 -20950.355,E2 -20950.355} C_VEL
LIN {X 0,Y 207.596,Z 341.164,A -85,B 0,C 180,E1 -20952.772,E2 -20952.772} C_VEL
LIN {X 0,Y 206.572,Z 347.972,A -85,B 0,C 180,E1 -20955.723,E2 -20955.723} C_VEL
LIN {X 0,Y 206.096,Z 354.687,A -85,B 0,C 180,E1 -20959.441,E2 -20959.441} C_VEL
LIN {X 0,Y 205.868,Z 362.208,A -85,B 0,C 180,E1 -20962.154,E2 -20962.154} C_VEL
LIN {X 0,Y 205.787,Z 368.848,A -85,B 0,C 180,E1 -20965.105,E2 -20965.105} C_VEL
LIN {X 0,Y 205.817,Z 374.084,A -85,B 0,C 180,E1 -20968.046,E2 -20968.046} C_VEL
LIN {X 0,Y 205.847,Z 376.863,A -85,B 0,C 180,E1 -20970.003,E2 -20970.003} C_VEL
LIN {X 0,Y 205.505,Z 379.082,A -85,B 0,C 180,E1 -20971.962,E2 -20971.962} C_VEL
LIN {X 0,Y 204.94,Z 382.325,A -85,B 0,C 180,E1 -20976.013,E2 -20976.013} C_VEL
LIN {X 0,Y 205.217,Z 383.97,A -85,B 0,C 180,E1 -20979.862,E2 -20979.862} C_VEL
LIN {X 0,Y 206.447,Z 384.331,A -85,B 0,C 180,E1 -20983.789,E2 -20983.789} C_VEL
LIN {X 0,Y 208.942,Z 383.422,A -85,B 0,C 180,E1 -20987.624,E2 -20987.624} C_VEL
LIN {X 0,Y 212.618,Z 381.248,A -85,B 0,C 180,E1 -20991.324,E2 -20991.324} C_VEL
LIN {X 0,Y 217.196,Z 377.818,A -85,B 0,C 180,E1 -20994.878,E2 -20994.878} C_VEL
LIN {X 0,Y 223.037,Z 373.035,A -85,B 0,C 180,E1 -20998.209,E2 -20998.209} C_VEL
LIN {X 0,Y 230.067,Z 366.832,A -85,B 0,C 180,E1 -21001.288,E2 -21001.288} C_VEL
LIN {X 0,Y 237.052,Z 360.042,A -85,B 0,C 180,E1 -21003.826,E2 -21003.826} C_VEL
LIN {X 0,Y 245.576,Z 350.838,A -85,B 0,C 180,E1 -21006.432,E2 -21006.432} C_VEL
LIN {X 0,Y 253.295,Z 341.287,A -85,B 0,C 180,E1 -21008.734,E2 -21008.734} C_VEL
LIN {X 0,Y 258.717,Z 333.343,A -85,B 0,C 180,E1 -21010.691,E2 -21010.691} C_VEL
LIN {X 0,Y 262.073,Z 328.013,A -85,B 0,C 180,E1 -21012.102,E2 -21012.102} C_VEL
LIN {X 0,Y 263.244,Z 326.055,A -85,B 0,C 180,E1 -21012.676,E2 -21012.676} C_VEL
LIN {X 0,Y 263.033,Z 325.258,A -85,B 0,C 180,E1 -21014.005,E2 -21014.005} C_VEL
LIN {X 0,Y 262.039,Z 325.534,A -85,B 0,C 180,E1 -21016.401,E2 -21016.401} C_VEL
LIN {X 0,Y 260.725,Z 327.1,A -85,B 0,C 180,E1 -21018.278,E2 -21018.278} C_VEL
LIN {X 0,Y 258.303,Z 330.617,A -85,B 0,C 180,E1 -21020.497,E2 -21020.497} C_VEL
LIN {X 0,Y 255.473,Z 335.155,A -85,B 0,C 180,E1 -21022.921,E2 -21022.921} C_VEL
LIN {X 0,Y 254.555,Z 336.519,A -85,B 0,C 180,E1 -21023.564,E2 -21023.564} C_VEL
LIN {X 0,Y 245.707,Z 345.922,A -85,B 0,C 180,E1 -21026.1,E2 -21026.1} C_VEL
LIN {X 0,Y 237.646,Z 353.34,A -85,B 0,C 180,E1 -21028.833,E2 -21028.833} C_VEL
LIN {X 0,Y 230.256,Z 359.143,A -85,B 0,C 180,E1 -21031.764,E2 -21031.764} C_VEL
LIN {X 0,Y 225.332,Z 362.491,A -85,B 0,C 180,E1 -21034.109,E2 -21034.109} C_VEL
LIN {X 0,Y 219.563,Z 365.697,A -85,B 0,C 180,E1 -21037.412,E2 -21037.412} C_VEL
LIN {X 0,Y 214.825,Z 367.57,A -85,B 0,C 180,E1 -21040.904,E2 -21040.904} C_VEL
LIN {X 0,Y 210.945,Z 368.109,A -85,B 0,C 180,E1 -21044.542,E2 -21044.542} C_VEL
LIN {X 0,Y 209.472,Z 367.866,A -85,B 0,C 180,E1 -21046.417,E2 -21046.417} C_VEL
LIN {X 0,Y 207.1,Z 366.622,A -85,B 0,C 180,E1 -21049.787,E2 -21049.787} C_VEL
LIN {X 0,Y 206.137,Z 365.143,A -85,B 0,C 180,E1 -21052.162,E2 -21052.162} C_VEL
LIN {X 0,Y 205.212,Z 361.538,A -85,B 0,C 180,E1 -21056.073,E2 -21056.073} C_VEL
LIN {X 0,Y 204.732,Z 356.374,A -85,B 0,C 180,E1 -21060,E2 -21060} C_VEL
LIN {X 0,Y 204.821,Z 351.342,A -85,B 0,C 180,E1 -21062.95,E2 -21062.95} C_VEL
LIN {X 0,Y 205.036,Z 344.302,A -85,B 0,C 180,E1 -21066.246,E2 -21066.246} C_VEL
LIN {X 0,Y 205.587,Z 336.108,A -85,B 0,C 180,E1 -21069.345,E2 -21069.345} C_VEL
LIN {X 0,Y 206.437,Z 326.578,A -85,B 0,C 180,E1 -21072.285,E2 -21072.285} C_VEL
LIN {X 0,Y 207.618,Z 314.869,A -85,B 0,C 180,E1 -21075.209,E2 -21075.209} C_VEL
LIN {X 0,Y 208.95,Z 302.773,A -85,B 0,C 180,E1 -21077.621,E2 -21077.621} C_VEL
LIN {X 0,Y 210.18,Z 289.783,A -85,B 0,C 180,E1 -21079.698,E2 -21079.698} C_VEL
LIN {X 0,Y 210.597,Z 285.699,A -85,B 0,C 180,E1 -21080.259,E2 -21080.259} C_VEL
LIN {X 0,Y 208.513,Z 270.982,A -85,B 0,C 180,E1 -21081.995,E2 -21081.995} C_VEL
LIN {X 0,Y 207.072,Z 257.22,A -85,B 0,C 180,E1 -21083.215,E2 -21083.215} C_VEL
LIN {X 0,Y 207.024,Z 256.162,A -85,B 0,C 180,E1 -21083.34,E2 -21083.34} C_VEL
LIN {X 0,Y 207.71,Z 247.135,A -85,B 0,C 180,E1 -21088.386,E2 -21088.386} C_VEL
LIN {X 0,Y 208.436,Z 239.566,A -85,B 0,C 180,E1 -21092.649,E2 -21092.649} C_VEL
LIN {X 0,Y 209.042,Z 233.285,A -85,B 0,C 180,E1 -21096.204,E2 -21096.204} C_VEL
LIN {X 0,Y 208.957,Z 229.833,A -85,B 0,C 180,E1 -21098.209,E2 -21098.209} C_VEL
LIN {X 0,Y 207.883,Z 223.61,A -85,B 0,C 180,E1 -21101.944,E2 -21101.944} C_VEL
LIN {X 0,Y 207.04,Z 219.298,A -85,B 0,C 180,E1 -21104.682,E2 -21104.682} C_VEL
LIN {X 0,Y 207.424,Z 221.473,A -85,B 0,C 180,E1 -21108.195,E2 -21108.195} C_VEL
LIN {X 0,Y 207.919,Z 224.388,A -85,B 0,C 180,E1 -21112.521,E2 -21112.521} C_VEL
LIN {X 0,Y 208.226,Z 226.178,A -85,B 0,C 180,E1 -21114.983,E2 -21114.983} C_VEL
LIN {X 0,Y 208.414,Z 228.087,A -85,B 0,C 180,E1 -21117.463,E2 -21117.463} C_VEL
LIN {X 0,Y 208.436,Z 231.723,A -85,B 0,C 180,E1 -21121.83,E2 -21121.83} C_VEL
LIN {X 0,Y 208.267,Z 234.07,A -85,B 0,C 180,E1 -21124.297,E2 -21124.297} C_VEL
LIN {X 0,Y 212.215,Z 245.005,A -85,B 0,C 180,E1 -21125.766,E2 -21125.766} C_VEL
LIN {X 0,Y 214.633,Z 253.58,A -85,B 0,C 180,E1 -21127.115,E2 -21127.115} C_VEL
LIN {X 0,Y 216.451,Z 262.782,A -85,B 0,C 180,E1 -21128.82,E2 -21128.82} C_VEL
LIN {X 0,Y 217.092,Z 269.079,A -85,B 0,C 180,E1 -21130.152,E2 -21130.152} C_VEL
LIN {X 0,Y 215.536,Z 277.298,A -85,B 0,C 180,E1 -21131.952,E2 -21131.952} C_VEL
LIN {X 0,Y 213.481,Z 285.272,A -85,B 0,C 180,E1 -21134.238,E2 -21134.238} C_VEL
LIN {X 0,Y 211.641,Z 291.36,A -85,B 0,C 180,E1 -21136.556,E2 -21136.556} C_VEL
LIN {X 0,Y 210.413,Z 295.209,A -85,B 0,C 180,E1 -21138.437,E2 -21138.437} C_VEL
LIN {X 0,Y 209.433,Z 299.522,A -85,B 0,C 180,E1 -21141.312,E2 -21141.312} C_VEL
LIN {X 0,Y 208.232,Z 302.487,A -85,B 0,C 180,E1 -21144.186,E2 -21144.186} C_VEL
LIN {X 0,Y 207.893,Z 303.726,A -85,B 0,C 180,E1 -21146.121,E2 -21146.121} C_VEL
LIN {X 0,Y 207.59,Z 304.486,A -85,B 0,C 180,E1 -21148.057,E2 -21148.057} C_VEL
LIN {X 0,Y 207.474,Z 304.758,A -85,B 0,C 180,E1 -21149.997,E2 -21149.997} C_VEL
LIN {X 0,Y 207.589,Z 304.519,A -85,B 0,C 180,E1 -21151.938,E2 -21151.938} C_VEL
LIN {X 0,Y 207.891,Z 303.805,A -85,B 0,C 180,E1 -21153.874,E2 -21153.874} C_VEL
LIN {X 0,Y 208.23,Z 302.611,A -85,B 0,C 180,E1 -21155.809,E2 -21155.809} C_VEL
LIN {X 0,Y 209.42,Z 299.697,A -85,B 0,C 180,E1 -21158.683,E2 -21158.683} C_VEL
LIN {X 0,Y 210.371,Z 295.473,A -85,B 0,C 180,E1 -21161.56,E2 -21161.56} C_VEL
LIN {X 0,Y 211.172,Z 293.652,A -85,B 0,C 180,E1 -21162.491,E2 -21162.491} C_VEL
LIN {X 0,Y 212.267,Z 289.475,A -85,B 0,C 180,E1 -21164.375,E2 -21164.375} C_VEL
LIN {X 0,Y 214.289,Z 282.804,A -85,B 0,C 180,E1 -21166.674,E2 -21166.674} C_VEL
LIN {X 0,Y 216.068,Z 274.957,A -85,B 0,C 180,E1 -21168.733,E2 -21168.733} C_VEL
LIN {X 0,Y 217.211,Z 267.871,A -85,B 0,C 180,E1 -21170.229,E2 -21170.229} C_VEL
LIN {X 0,Y 216.109,Z 260.437,A -85,B 0,C 180,E1 -21171.795,E2 -21171.795} C_VEL
LIN {X 0,Y 213.989,Z 250.906,A -85,B 0,C 180,E1 -21173.469,E2 -21173.469} C_VEL
LIN {X 0,Y 210.967,Z 241.364,A -85,B 0,C 180,E1 -21174.912,E2 -21174.912} C_VEL
LIN {X 0,Y 208.257,Z 233.942,A -85,B 0,C 180,E1 -21175.894,E2 -21175.894} C_VEL
LIN {X 0,Y 208.447,Z 231.386,A -85,B 0,C 180,E1 -21178.763,E2 -21178.763} C_VEL
LIN {X 0,Y 208.401,Z 228.156,A -85,B 0,C 180,E1 -21182.651,E2 -21182.651} C_VEL
LIN {X 0,Y 208.181,Z 225.714,A -85,B 0,C 180,E1 -21185.882,E2 -21185.882} C_VEL
LIN {X 0,Y 207.66,Z 222.836,A -85,B 0,C 180,E1 -21190.014,E2 -21190.014} C_VEL
LIN {X 0,Y 207.106,Z 219.893,A -85,B 0,C 180,E1 -21194.551,E2 -21194.551} C_VEL
LIN {X 0,Y 206.686,Z 217.736,A -85,B 0,C 180,E1 -21198.419,E2 -21198.419} C_VEL
LIN {X 0,Y 206.692,Z 217.731,A -85,B 0,C 180,E1 -21202.262,E2 -21202.262} C_VEL
LIN {X 0,Y 206.698,Z 217.729,A -85,B 0,C 180,E1 -21207.042,E2 -21207.042} C_VEL
LIN {X 0,Y 206.758,Z 217.728,A -85,B 0,C 180,E1 -21212.095,E2 -21212.095} C_VEL
LIN {X 0,Y 206.776,Z 217.724,A -85,B 0,C 180,E1 -21216.583,E2 -21216.583} C_VEL
LIN {X 0,Y 206.864,Z 217.718,A -85,B 0,C 180,E1 -21222.196,E2 -21222.196} C_VEL
LIN {X 0,Y 206.886,Z 217.705,A -85,B 0,C 180,E1 -21226.244,E2 -21226.244} C_VEL
LIN {X 0,Y 207.09,Z 217.671,A -85,B 0,C 180,E1 -21230.23,E2 -21230.23} C_VEL
LIN {X 0,Y 207.055,Z 217.68,A -85,B 0,C 180,E1 -21234.155,E2 -21234.155} C_VEL
LIN {X 0,Y 207.372,Z 217.652,A -85,B 0,C 180,E1 -21238.058,E2 -21238.058} C_VEL
LIN {X 0,Y 207.505,Z 217.62,A -85,B 0,C 180,E1 -21240,E2 -21240} C_VEL
LIN {X 0,Y 207.371,Z 217.651,A -85,B 0,C 180,E1 -21241.942,E2 -21241.942} C_VEL
LIN {X 0,Y 207.168,Z 217.675,A -85,B 0,C 180,E1 -21247.799,E2 -21247.799} C_VEL
LIN {X 0,Y 206.929,Z 217.709,A -85,B 0,C 180,E1 -21251.758,E2 -21251.758} C_VEL
LIN {X 0,Y 206.82,Z 217.724,A -85,B 0,C 180,E1 -21255.774,E2 -21255.774} C_VEL
LIN {X 0,Y 206.705,Z 217.739,A -85,B 0,C 180,E1 -21259.877,E2 -21259.877} C_VEL
LIN {X 0,Y 206.734,Z 217.821,A -85,B 0,C 180,E1 -21262.71,E2 -21262.71} C_VEL
LIN {X 0,Y 207.89,Z 222.455,A -85,B 0,C 180,E1 -21268.248,E2 -21268.248} C_VEL
LIN {X 0,Y 209.02,Z 226.999,A -85,B 0,C 180,E1 -21272.803,E2 -21272.803} C_VEL
LIN {X 0,Y 210.137,Z 231.679,A -85,B 0,C 180,E1 -21277.014,E2 -21277.014} C_VEL
LIN {X 0,Y 211.423,Z 237.55,A -85,B 0,C 180,E1 -21281.669,E2 -21281.669} C_VEL
LIN {X 0,Y 212.885,Z 244.434,A -85,B 0,C 180,E1 -21286.576,E2 -21286.576} C_VEL
LIN {X 0,Y 214.083,Z 250.174,A -85,B 0,C 180,E1 -21290.331,E2 -21290.331} C_VEL
LIN {X 0,Y 215.257,Z 256.103,A -85,B 0,C 180,E1 -21294.01,E2 -21294.01} C_VEL
LIN {X 0,Y 214.407,Z 258.771,A -85,B 0,C 180,E1 -21295.451,E2 -21295.451} C_VEL
LIN {X 0,Y 211.576,Z 266.076,A -85,B 0,C 180,E1 -21299.321,E2 -21299.321} C_VEL
LIN {X 0,Y 212.721,Z 278.437,A -85,B 0,C 180,E1 -21300.336,E2 -21300.336} C_VEL
LIN {X 0,Y 213.137,Z 290.945,A -85,B 0,C 180,E1 -21301.709,E2 -21301.709} C_VEL
LIN {X 0,Y 212.86,Z 301.326,A -85,B 0,C 180,E1 -21303.142,E2 -21303.142} C_VEL
LIN {X 0,Y 212.231,Z 309.612,A -85,B 0,C 180,E1 -21304.514,E2 -21304.514} C_VEL
LIN {X 0,Y 211.243,Z 314.528,A -85,B 0,C 180,E1 -21305.417,E2 -21305.417} C_VEL
LIN {X 0,Y 209.269,Z 319.148,A -85,B 0,C 180,E1 -21306.278,E2 -21306.278} C_VEL
LIN {X 0,Y 203.754,Z 329.15,A -85,B 0,C 180,E1 -21308.506,E2 -21308.506} C_VEL
LIN {X 0,Y 202.259,Z 333.116,A -85,B 0,C 180,E1 -21309.692,E2 -21309.692} C_VEL
LIN {X 0,Y 200.775,Z 340.134,A -85,B 0,C 180,E1 -21312.167,E2 -21312.167} C_VEL
LIN {X 0,Y 199.593,Z 346.956,A -85,B 0,C 180,E1 -21315.212,E2 -21315.212} C_VEL
LIN {X 0,Y 199.05,Z 353.081,A -85,B 0,C 180,E1 -21318.805,E2 -21318.805} C_VEL
LIN {X 0,Y 199.026,Z 355.079,A -85,B 0,C 180,E1 -21320.116,E2 -21320.116} C_VEL
LIN {X 0,Y 198.852,Z 363.09,A -85,B 0,C 180,E1 -21323.206,E2 -21323.206} C_VEL
LIN {X 0,Y 198.817,Z 368.808,A -85,B 0,C 180,E1 -21325.949,E2 -21325.949} C_VEL
LIN {X 0,Y 198.904,Z 373.891,A -85,B 0,C 180,E1 -21328.99,E2 -21328.99} C_VEL
LIN {X 0,Y 198.735,Z 376.521,A -85,B 0,C 180,E1 -21331.016,E2 -21331.016} C_VEL
LIN {X 0,Y 198.148,Z 379.566,A -85,B 0,C 180,E1 -21334.07,E2 -21334.07} C_VEL
LIN {X 0,Y 197.963,Z 382.241,A -85,B 0,C 180,E1 -21338.167,E2 -21338.167} C_VEL
LIN {X 0,Y 198.751,Z 383.571,A -85,B 0,C 180,E1 -21342.252,E2 -21342.252} C_VEL
LIN {X 0,Y 200.665,Z 383.635,A -85,B 0,C 180,E1 -21346.274,E2 -21346.274} C_VEL
LIN {X 0,Y 203.955,Z 382.448,A -85,B 0,C 180,E1 -21350.159,E2 -21350.159} C_VEL
LIN {X 0,Y 208.26,Z 379.995,A -85,B 0,C 180,E1 -21353.891,E2 -21353.891} C_VEL
LIN {X 0,Y 213.641,Z 376.326,A -85,B 0,C 180,E1 -21357.425,E2 -21357.425} C_VEL
LIN {X 0,Y 220.37,Z 371.343,A -85,B 0,C 180,E1 -21360.684,E2 -21360.684} C_VEL
LIN {X 0,Y 228.1,Z 364.93,A -85,B 0,C 180,E1 -21363.686,E2 -21363.686} C_VEL
LIN {X 0,Y 236.731,Z 356.953,A -85,B 0,C 180,E1 -21366.426,E2 -21366.426} C_VEL
LIN {X 0,Y 245.812,Z 347.416,A -85,B 0,C 180,E1 -21368.979,E2 -21368.979} C_VEL
LIN {X 0,Y 250.932,Z 341.29,A -85,B 0,C 180,E1 -21370.5,E2 -21370.5} C_VEL
LIN {X 0,Y 256.858,Z 333.342,A -85,B 0,C 180,E1 -21372.626,E2 -21372.626} C_VEL
LIN {X 0,Y 257.734,Z 332.121,A -85,B 0,C 180,E1 -21372.98,E2 -21372.98} C_VEL
LIN {X 0,Y 258.463,Z 330.794,A -85,B 0,C 180,E1 -21373.708,E2 -21373.708} C_VEL
LIN {X 0,Y 257.886,Z 330.684,A -85,B 0,C 180,E1 -21375.12,E2 -21375.12} C_VEL
LIN {X 0,Y 256.89,Z 331.304,A -85,B 0,C 180,E1 -21376.847,E2 -21376.847} C_VEL
LIN {X 0,Y 256.144,Z 332.099,A -85,B 0,C 180,E1 -21377.804,E2 -21377.804} C_VEL
LIN {X 0,Y 253.045,Z 335.866,A -85,B 0,C 180,E1 -21380.298,E2 -21380.298} C_VEL
LIN {X 0,Y 249.855,Z 339.989,A -85,B 0,C 180,E1 -21382.584,E2 -21382.584} C_VEL
LIN {X 0,Y 242.442,Z 347.136,A -85,B 0,C 180,E1 -21384.566,E2 -21384.566} C_VEL
LIN {X 0,Y 233.753,Z 354.528,A -85,B 0,C 180,E1 -21387.339,E2 -21387.339} C_VEL
LIN {X 0,Y 226.091,Z 360.012,A -85,B 0,C 180,E1 -21390.175,E2 -21390.175} C_VEL
LIN {X 0,Y 219.148,Z 364.201,A -85,B 0,C 180,E1 -21393.322,E2 -21393.322} C_VEL
LIN {X 0,Y 213.138,Z 366.979,A -85,B 0,C 180,E1 -21396.691,E2 -21396.691} C_VEL
LIN {X 0,Y 208.19,Z 368.432,A -85,B 0,C 180,E1 -21400.271,E2 -21400.271} C_VEL
LIN {X 0,Y 204.128,Z 368.624,A -85,B 0,C 180,E1 -21404.012,E2 -21404.012} C_VEL
LIN {X 0,Y 202.599,Z 368.221,A -85,B 0,C 180,E1 -21405.947,E2 -21405.947} C_VEL
LIN {X 0,Y 201.017,Z 367.478,A -85,B 0,C 180,E1 -21407.891,E2 -21407.891} C_VEL
LIN {X 0,Y 199.111,Z 364.955,A -85,B 0,C 180,E1 -21411.884,E2 -21411.884} C_VEL
LIN {X 0,Y 198.162,Z 361.058,A -85,B 0,C 180,E1 -21415.933,E2 -21415.933} C_VEL
LIN {X 0,Y 197.712,Z 357.075,A -85,B 0,C 180,E1 -21418.982,E2 -21418.982} C_VEL
LIN {X 0,Y 197.72,Z 352.128,A -85,B 0,C 180,E1 -21422.037,E2 -21422.037} C_VEL
LIN {X 0,Y 197.914,Z 344.874,A -85,B 0,C 180,E1 -21425.612,E2 -21425.612} C_VEL
LIN {X 0,Y 198.397,Z 337.202,A -85,B 0,C 180,E1 -21428.659,E2 -21428.659} C_VEL
LIN {X 0,Y 199.217,Z 327.896,A -85,B 0,C 180,E1 -21431.704,E2 -21431.704} C_VEL
LIN {X 0,Y 200.185,Z 317.456,A -85,B 0,C 180,E1 -21434.486,E2 -21434.486} C_VEL
LIN {X 0,Y 201.28,Z 307.217,A -85,B 0,C 180,E1 -21436.742,E2 -21436.742} C_VEL
LIN {X 0,Y 202.39,Z 296.314,A -85,B 0,C 180,E1 -21438.736,E2 -21438.736} C_VEL
LIN {X 0,Y 203.429,Z 286.561,A -85,B 0,C 180,E1 -21440.211,E2 -21440.211} C_VEL
LIN {X 0,Y 201.573,Z 272.56,A -85,B 0,C 180,E1 -21441.944,E2 -21441.944} C_VEL
LIN {X 0,Y 200.065,Z 258.772,A -85,B 0,C 180,E1 -21443.251,E2 -21443.251} C_VEL
LIN {X 0,Y 199.97,Z 256.469,A -85,B 0,C 180,E1 -21443.5,E2 -21443.5} C_VEL
LIN {X 0,Y 200.715,Z 247.017,A -85,B 0,C 180,E1 -21448.907,E2 -21448.907} C_VEL
LIN {X 0,Y 201.592,Z 238.338,A -85,B 0,C 180,E1 -21453.904,E2 -21453.904} C_VEL
LIN {X 0,Y 202.039,Z 233.25,A -85,B 0,C 180,E1 -21456.86,E2 -21456.86} C_VEL
LIN {X 0,Y 201.527,Z 228.224,A -85,B 0,C 180,E1 -21459.892,E2 -21459.892} C_VEL
LIN {X 0,Y 200.172,Z 221.123,A -85,B 0,C 180,E1 -21464.395,E2 -21464.395} C_VEL
LIN {X 0,Y 200.607,Z 223.424,A -85,B 0,C 180,E1 -21468.266,E2 -21468.266} C_VEL
LIN {X 0,Y 200.914,Z 225.182,A -85,B 0,C 180,E1 -21470.973,E2 -21470.973} C_VEL
LIN {X 0,Y 201.18,Z 226.955,A -85,B 0,C 180,E1 -21473.565,E2 -21473.565} C_VEL
LIN {X 0,Y 201.45,Z 229.351,A -85,B 0,C 180,E1 -21476.855,E2 -21476.855} C_VEL
LIN {X 0,Y 201.534,Z 232.5,A -85,B 0,C 180,E1 -21480.774,E2 -21480.774} C_VEL
LIN {X 0,Y 201.372,Z 234.614,A -85,B 0,C 180,E1 -21483.207,E2 -21483.207} C_VEL
LIN {X 0,Y 205.276,Z 245.221,A -85,B 0,C 180,E1 -21484.729,E2 -21484.729} C_VEL
LIN {X 0,Y 208.052,Z 254.989,A -85,B 0,C 180,E1 -21486.35,E2 -21486.35} C_VEL
LIN {X 0,Y 209.849,Z 264.059,A -85,B 0,C 180,E1 -21488.123,E2 -21488.123} C_VEL
LIN {X 0,Y 210.499,Z 270.419,A -85,B 0,C 180,E1 -21489.542,E2 -21489.542} C_VEL
LIN {X 0,Y 208.88,Z 278.363,A -85,B 0,C 180,E1 -21491.357,E2 -21491.357} C_VEL
LIN {X 0,Y 206.733,Z 286.298,A -85,B 0,C 180,E1 -21493.71,E2 -21493.71} C_VEL
LIN {X 0,Y 204.812,Z 292.359,A -85,B 0,C 180,E1 -21496.099,E2 -21496.099} C_VEL
LIN {X 0,Y 203.531,Z 296.196,A -85,B 0,C 180,E1 -21498.04,E2 -21498.04} C_VEL
LIN {X 0,Y 202.488,Z 300.499,A -85,B 0,C 180,E1 -21501.012,E2 -21501.012} C_VEL
LIN {X 0,Y 201.242,Z 303.463,A -85,B 0,C 180,E1 -21503.984,E2 -21503.984} C_VEL
LIN {X 0,Y 200.882,Z 304.699,A -85,B 0,C 180,E1 -21505.985,E2 -21505.985} C_VEL
LIN {X 0,Y 200.567,Z 305.46,A -85,B 0,C 180,E1 -21507.989,E2 -21507.989} C_VEL
LIN {X 0,Y 200.446,Z 305.732,A -85,B 0,C 180,E1 -21509.997,E2 -21509.997} C_VEL
LIN {X 0,Y 200.565,Z 305.494,A -85,B 0,C 180,E1 -21512.005,E2 -21512.005} C_VEL
LIN {X 0,Y 200.88,Z 304.779,A -85,B 0,C 180,E1 -21514.01,E2 -21514.01} C_VEL
LIN {X 0,Y 201.24,Z 303.585,A -85,B 0,C 180,E1 -21516.011,E2 -21516.011} C_VEL
LIN {X 0,Y 202.474,Z 300.675,A -85,B 0,C 180,E1 -21518.984,E2 -21518.984} C_VEL
LIN {X 0,Y 203.488,Z 296.46,A -85,B 0,C 180,E1 -21521.957,E2 -21521.957} C_VEL
LIN {X 0,Y 204.315,Z 294.644,A -85,B 0,C 180,E1 -21522.917,E2 -21522.917} C_VEL
LIN {X 0,Y 205.468,Z 290.481,A -85,B 0,C 180,E1 -21524.862,E2 -21524.862} C_VEL
LIN {X 0,Y 207.575,Z 283.834,A -85,B 0,C 180,E1 -21527.23,E2 -21527.23} C_VEL
LIN {X 0,Y 209.442,Z 276.046,A -85,B 0,C 180,E1 -21529.349,E2 -21529.349} C_VEL
LIN {X 0,Y 210.571,Z 269.26,A -85,B 0,C 180,E1 -21530.848,E2 -21530.848} C_VEL
LIN {X 0,Y 209.536,Z 261.76,A -85,B 0,C 180,E1 -21532.504,E2 -21532.504} C_VEL
LIN {X 0,Y 207.446,Z 252.232,A -85,B 0,C 180,E1 -21534.272,E2 -21534.272} C_VEL
LIN {X 0,Y 204.336,Z 242.467,A -85,B 0,C 180,E1 -21535.848,E2 -21535.848} C_VEL
LIN {X 0,Y 201.395,Z 234.617,A -85,B 0,C 180,E1 -21536.975,E2 -21536.975} C_VEL
LIN {X 0,Y 201.539,Z 232.591,A -85,B 0,C 180,E1 -21539.332,E2 -21539.332} C_VEL
LIN {X 0,Y 201.427,Z 228.94,A -85,B 0,C 180,E1 -21543.932,E2 -21543.932} C_VEL
LIN {X 0,Y 201.207,Z 227.052,A -85,B 0,C 180,E1 -21546.546,E2 -21546.546} C_VEL
LIN {X 0,Y 200.853,Z 224.915,A -85,B 0,C 180,E1 -21549.664,E2 -21549.664} C_VEL
LIN {X 0,Y 200.304,Z 221.871,A -85,B 0,C 180,E1 -21554.562,E2 -21554.562} C_VEL
LIN {X 0,Y 199.905,Z 219.852,A -85,B 0,C 180,E1 -21558.089,E2 -21558.089} C_VEL
LIN {X 0,Y 199.636,Z 218.617,A -85,B 0,C 180,E1 -21560.754,E2 -21560.754} C_VEL
LIN {X 0,Y 199.616,Z 218.611,A -85,B 0,C 180,E1 -21565.714,E2 -21565.714} C_VEL
LIN {X 0,Y 199.695,Z 218.611,A -85,B 0,C 180,E1 -21568.136,E2 -21568.136} C_VEL
LIN {X 0,Y 199.679,Z 218.613,A -85,B 0,C 180,E1 -21572.77,E2 -21572.77} C_VEL
LIN {X 0,Y 199.731,Z 218.607,A -85,B 0,C 180,E1 -21577.228,E2 -21577.228} C_VEL
LIN {X 0,Y 199.788,Z 218.597,A -85,B 0,C 180,E1 -21581.756,E2 -21581.756} C_VEL
LIN {X 0,Y 199.826,Z 218.579,A -85,B 0,C 180,E1 -21585.747,E2 -21585.747} C_VEL
LIN {X 0,Y 200.013,Z 218.553,A -85,B 0,C 180,E1 -21589.881,E2 -21589.881} C_VEL
LIN {X 0,Y 200.017,Z 218.558,A -85,B 0,C 180,E1 -21593.949,E2 -21593.949} C_VEL
LIN {X 0,Y 200.311,Z 218.532,A -85,B 0,C 180,E1 -21597.989,E2 -21597.989} C_VEL
LIN {X 0,Y 200.469,Z 218.496,A -85,B 0,C 180,E1 -21600,E2 -21600} C_VEL
LIN {X 0,Y 200.017,Z 218.558,A -85,B 0,C 180,E1 -21604.03,E2 -21604.03} C_VEL
LIN {X 0,Y 200.109,Z 218.551,A -85,B 0,C 180,E1 -21608.076,E2 -21608.076} C_VEL
LIN {X 0,Y 199.871,Z 218.583,A -85,B 0,C 180,E1 -21612.18,E2 -21612.18} C_VEL
LIN {X 0,Y 199.755,Z 218.598,A -85,B 0,C 180,E1 -21616.348,E2 -21616.348} C_VEL
LIN {X 0,Y 199.661,Z 218.624,A -85,B 0,C 180,E1 -21620.072,E2 -21620.072} C_VEL
LIN {X 0,Y 200.356,Z 221.624,A -85,B 0,C 180,E1 -21624.222,E2 -21624.222} C_VEL
LIN {X 0,Y 201.471,Z 225.947,A -85,B 0,C 180,E1 -21629.304,E2 -21629.304} C_VEL
LIN {X 0,Y 202.607,Z 230.349,A -85,B 0,C 180,E1 -21633.711,E2 -21633.711} C_VEL
LIN {X 0,Y 203.778,Z 235.584,A -85,B 0,C 180,E1 -21638.374,E2 -21638.374} C_VEL
LIN {X 0,Y 204.715,Z 240.124,A -85,B 0,C 180,E1 -21642.023,E2 -21642.023} C_VEL
LIN {X 0,Y 206.377,Z 247.732,A -85,B 0,C 180,E1 -21647.581,E2 -21647.581} C_VEL
LIN {X 0,Y 207.862,Z 255.179,A -85,B 0,C 180,E1 -21652.516,E2 -21652.516} C_VEL
LIN {X 0,Y 208.135,Z 257.802,A -85,B 0,C 180,E1 -21654.135,E2 -21654.135} C_VEL
LIN {X 0,Y 205.018,Z 265.401,A -85,B 0,C 180,E1 -21658.339,E2 -21658.339} C_VEL
LIN {X 0,Y 206.182,Z 277.426,A -85,B 0,C 180,E1 -21659.374,E2 -21659.374} C_VEL
LIN {X 0,Y 206.513,Z 289.515,A -85,B 0,C 180,E1 -21660.731,E2 -21660.731} C_VEL
LIN {X 0,Y 206.328,Z 299.926,A -85,B 0,C 180,E1 -21662.205,E2 -21662.205} C_VEL
LIN {X 0,Y 205.371,Z 310.91,A -85,B 0,C 180,E1 -21664.134,E2 -21664.134} C_VEL
LIN {X 0,Y 204.704,Z 319.28,A -85,B 0,C 180,E1 -21665.943,E2 -21665.943} C_VEL
LIN {X 0,Y 204.189,Z 324.532,A -85,B 0,C 180,E1 -21667.222,E2 -21667.222} C_VEL
LIN {X 0,Y 202.259,Z 333.116,A -85,B 0,C 180,E1 -21669.692,E2 -21669.692} C_VEL
LIN {X 0,Y 200.768,Z 336.931,A -85,B 0,C 180,E1 -21670.943,E2 -21670.943} C_VEL
LIN {X 0,Y 196.781,Z 342.439,A -85,B 0,C 180,E1 -21673.034,E2 -21673.034} C_VEL
LIN {X 0,Y 193.119,Z 347.188,A -85,B 0,C 180,E1 -21675.334,E2 -21675.334} C_VEL
LIN {X 0,Y 192.146,Z 349.77,A -85,B 0,C 180,E1 -21676.869,E2 -21676.869} C_VEL
LIN {X 0,Y 191.945,Z 353.482,A -85,B 0,C 180,E1 -21679.454,E2 -21679.454} C_VEL
LIN {X 0,Y 192.022,Z 355.126,A -85,B 0,C 180,E1 -21680.749,E2 -21680.749} C_VEL
LIN {X 0,Y 191.902,Z 362.419,A -85,B 0,C 180,E1 -21683.695,E2 -21683.695} C_VEL
LIN {X 0,Y 191.915,Z 368.677,A -85,B 0,C 180,E1 -21686.854,E2 -21686.854} C_VEL
LIN {X 0,Y 191.991,Z 373.604,A -85,B 0,C 180,E1 -21690.003,E2 -21690.003} C_VEL
LIN {X 0,Y 191.381,Z 377.199,A -85,B 0,C 180,E1 -21693.16,E2 -21693.16} C_VEL
LIN {X 0,Y 190.973,Z 379.91,A -85,B 0,C 180,E1 -21696.471,E2 -21696.471} C_VEL
LIN {X 0,Y 191.292,Z 382.116,A -85,B 0,C 180,E1 -21700.588,E2 -21700.588} C_VEL
LIN {X 0,Y 192.656,Z 383.092,A -85,B 0,C 180,E1 -21704.797,E2 -21704.797} C_VEL
LIN {X 0,Y 195.459,Z 382.852,A -85,B 0,C 180,E1 -21708.884,E2 -21708.884} C_VEL
LIN {X 0,Y 199.459,Z 381.393,A -85,B 0,C 180,E1 -21712.807,E2 -21712.807} C_VEL
LIN {X 0,Y 204.441,Z 378.747,A -85,B 0,C 180,E1 -21716.547,E2 -21716.547} C_VEL
LIN {X 0,Y 210.756,Z 374.888,A -85,B 0,C 180,E1 -21720.016,E2 -21720.016} C_VEL
LIN {X 0,Y 218.258,Z 369.707,A -85,B 0,C 180,E1 -21723.192,E2 -21723.192} C_VEL
LIN {X 0,Y 226.655,Z 363.12,A -85,B 0,C 180,E1 -21726.099,E2 -21726.099} C_VEL
LIN {X 0,Y 235.944,Z 355.006,A -85,B 0,C 180,E1 -21728.723,E2 -21728.723} C_VEL
LIN {X 0,Y 245.258,Z 345.578,A -85,B 0,C 180,E1 -21731.232,E2 -21731.232} C_VEL
LIN {X 0,Y 251.471,Z 338.364,A -85,B 0,C 180,E1 -21733.217,E2 -21733.217} C_VEL
LIN {X 0,Y 253.335,Z 336.087,A -85,B 0,C 180,E1 -21733.914,E2 -21733.914} C_VEL
LIN {X 0,Y 252.12,Z 336.314,A -85,B 0,C 180,E1 -21736.452,E2 -21736.452} C_VEL
LIN {X 0,Y 250.842,Z 337.479,A -85,B 0,C 180,E1 -21737.745,E2 -21737.745} C_VEL
LIN {X 0,Y 247.636,Z 340.77,A -85,B 0,C 180,E1 -21740.023,E2 -21740.023} C_VEL
LIN {X 0,Y 246.084,Z 342.43,A -85,B 0,C 180,E1 -21741.075,E2 -21741.075} C_VEL
LIN {X 0,Y 244.738,Z 343.813,A -85,B 0,C 180,E1 -21741.662,E2 -21741.662} C_VEL
LIN {X 0,Y 237.113,Z 350.373,A -85,B 0,C 180,E1 -21743.644,E2 -21743.644} C_VEL
LIN {X 0,Y 228.319,Z 356.987,A -85,B 0,C 180,E1 -21746.353,E2 -21746.353} C_VEL
LIN {X 0,Y 220.194,Z 362.116,A -85,B 0,C 180,E1 -21749.291,E2 -21749.291} C_VEL
LIN {X 0,Y 212.981,Z 365.802,A -85,B 0,C 180,E1 -21752.485,E2 -21752.485} C_VEL
LIN {X 0,Y 206.738,Z 368.175,A -85,B 0,C 180,E1 -21755.925,E2 -21755.925} C_VEL
LIN {X 0,Y 201.571,Z 369.239,A -85,B 0,C 180,E1 -21759.595,E2 -21759.595} C_VEL
LIN {X 0,Y 197.346,Z 369.026,A -85,B 0,C 180,E1 -21763.447,E2 -21763.447} C_VEL
LIN {X 0,Y 195.728,Z 368.434,A -85,B 0,C 180,E1 -21765.443,E2 -21765.443} C_VEL
LIN {X 0,Y 194.09,Z 367.524,A -85,B 0,C 180,E1 -21767.452,E2 -21767.452} C_VEL
LIN {X 0,Y 192.093,Z 364.702,A -85,B 0,C 180,E1 -21771.585,E2 -21771.585} C_VEL
LIN {X 0,Y 191.114,Z 360.439,A -85,B 0,C 180,E1 -21775.782,E2 -21775.782} C_VEL
LIN {X 0,Y 190.617,Z 354.607,A -85,B 0,C 180,E1 -21780,E2 -21780} C_VEL
LIN {X 0,Y 190.763,Z 347.944,A -85,B 0,C 180,E1 -21783.697,E2 -21783.697} C_VEL
LIN {X 0,Y 191.158,Z 339.588,A -85,B 0,C 180,E1 -21787.392,E2 -21787.392} C_VEL
LIN {X 0,Y 191.855,Z 330.722,A -85,B 0,C 180,E1 -21790.554,E2 -21790.554} C_VEL
LIN {X 0,Y 192.825,Z 319.904,A -85,B 0,C 180,E1 -21793.704,E2 -21793.704} C_VEL
LIN {X 0,Y 194.008,Z 308.902,A -85,B 0,C 180,E1 -21796.305,E2 -21796.305} C_VEL
LIN {X 0,Y 195.251,Z 296.88,A -85,B 0,C 180,E1 -21798.63,E2 -21798.63} C_VEL
LIN {X 0,Y 196.245,Z 287.155,A -85,B 0,C 180,E1 -21800.163,E2 -21800.163} C_VEL
LIN {X 0,Y 195.531,Z 280.551,A -85,B 0,C 180,E1 -21801.065,E2 -21801.065} C_VEL
LIN {X 0,Y 193.727,Z 266.583,A -85,B 0,C 180,E1 -21802.672,E2 -21802.672} C_VEL
LIN {X 0,Y 192.888,Z 256.926,A -85,B 0,C 180,E1 -21803.557,E2 -21803.557} C_VEL
LIN {X 0,Y 193.641,Z 247.947,A -85,B 0,C 180,E1 -21808.814,E2 -21808.814} C_VEL
LIN {X 0,Y 194.511,Z 239.503,A -85,B 0,C 180,E1 -21813.792,E2 -21813.792} C_VEL
LIN {X 0,Y 195.006,Z 233.211,A -85,B 0,C 180,E1 -21817.541,E2 -21817.541} C_VEL
LIN {X 0,Y 194.12,Z 227.132,A -85,B 0,C 180,E1 -21821.327,E2 -21821.327} C_VEL
LIN {X 0,Y 193.312,Z 222.935,A -85,B 0,C 180,E1 -21824.112,E2 -21824.112} C_VEL
LIN {X 0,Y 193.582,Z 224.321,A -85,B 0,C 180,E1 -21826.561,E2 -21826.561} C_VEL
LIN {X 0,Y 193.855,Z 226.167,A -85,B 0,C 180,E1 -21829.582,E2 -21829.582} C_VEL
LIN {X 0,Y 194.203,Z 228.26,A -85,B 0,C 180,E1 -21832.765,E2 -21832.765} C_VEL
LIN {X 0,Y 194.582,Z 231.4,A -85,B 0,C 180,E1 -21837.193,E2 -21837.193} C_VEL
LIN {X 0,Y 194.596,Z 233.664,A -85,B 0,C 180,E1 -21840.087,E2 -21840.087} C_VEL
LIN {X 0,Y 194.554,Z 235.524,A -85,B 0,C 180,E1 -21842.096,E2 -21842.096} C_VEL
LIN {X 0,Y 198.278,Z 245.348,A -85,B 0,C 180,E1 -21843.587,E2 -21843.587} C_VEL
LIN {X 0,Y 201.127,Z 254.595,A -85,B 0,C 180,E1 -21845.206,E2 -21845.206} C_VEL
LIN {X 0,Y 203.013,Z 263.923,A -85,B 0,C 180,E1 -21847.082,E2 -21847.082} C_VEL
LIN {X 0,Y 203.926,Z 271.748,A -85,B 0,C 180,E1 -21848.889,E2 -21848.889} C_VEL
LIN {X 0,Y 202.248,Z 279.422,A -85,B 0,C 180,E1 -21850.721,E2 -21850.721} C_VEL
LIN {X 0,Y 200.005,Z 287.321,A -85,B 0,C 180,E1 -21853.146,E2 -21853.146} C_VEL
LIN {X 0,Y 197.997,Z 293.361,A -85,B 0,C 180,E1 -21855.611,E2 -21855.611} C_VEL
LIN {X 0,Y 196.659,Z 297.185,A -85,B 0,C 180,E1 -21857.616,E2 -21857.616} C_VEL
LIN {X 0,Y 195.549,Z 301.476,A -85,B 0,C 180,E1 -21860.69,E2 -21860.69} C_VEL
LIN {X 0,Y 194.255,Z 304.439,A -85,B 0,C 180,E1 -21863.766,E2 -21863.766} C_VEL
LIN {X 0,Y 193.873,Z 305.674,A -85,B 0,C 180,E1 -21865.84,E2 -21865.84} C_VEL
LIN {X 0,Y 193.543,Z 306.434,A -85,B 0,C 180,E1 -21867.916,E2 -21867.916} C_VEL
LIN {X 0,Y 193.419,Z 306.707,A -85,B 0,C 180,E1 -21869.997,E2 -21869.997} C_VEL
LIN {X 0,Y 193.542,Z 306.467,A -85,B 0,C 180,E1 -21872.078,E2 -21872.078} C_VEL
LIN {X 0,Y 193.871,Z 305.753,A -85,B 0,C 180,E1 -21874.155,E2 -21874.155} C_VEL
LIN {X 0,Y 194.252,Z 304.559,A -85,B 0,C 180,E1 -21876.228,E2 -21876.228} C_VEL
LIN {X 0,Y 195.535,Z 301.65,A -85,B 0,C 180,E1 -21879.305,E2 -21879.305} C_VEL
LIN {X 0,Y 196.616,Z 297.447,A -85,B 0,C 180,E1 -21882.382,E2 -21882.382} C_VEL
LIN {X 0,Y 197.47,Z 295.636,A -85,B 0,C 180,E1 -21883.373,E2 -21883.373} C_VEL
LIN {X 0,Y 198.686,Z 291.487,A -85,B 0,C 180,E1 -21885.382,E2 -21885.382} C_VEL
LIN {X 0,Y 200.883,Z 284.862,A -85,B 0,C 180,E1 -21887.823,E2 -21887.823} C_VEL
LIN {X 0,Y 202.839,Z 277.137,A -85,B 0,C 180,E1 -21890.005,E2 -21890.005} C_VEL
LIN {X 0,Y 203.961,Z 270.637,A -85,B 0,C 180,E1 -21891.509,E2 -21891.509} C_VEL
LIN {X 0,Y 202.954,Z 263.081,A -85,B 0,C 180,E1 -21893.261,E2 -21893.261} C_VEL
LIN {X 0,Y 201.333,Z 255.268,A -85,B 0,C 180,E1 -21894.825,E2 -21894.825} C_VEL
LIN {X 0,Y 198.69,Z 246.337,A -85,B 0,C 180,E1 -21896.399,E2 -21896.399} C_VEL
LIN {X 0,Y 194.524,Z 235.295,A -85,B 0,C 180,E1 -21898.145,E2 -21898.145} C_VEL
LIN {X 0,Y 194.618,Z 233.49,A -85,B 0,C 180,E1 -21900.365,E2 -21900.365} C_VEL
LIN {X 0,Y 194.563,Z 230.801,A -85,B 0,C 180,E1 -21903.818,E2 -21903.818} C_VEL
LIN {X 0,Y 194.179,Z 227.91,A -85,B 0,C 180,E1 -21907.969,E2 -21907.969} C_VEL
LIN {X 0,Y 193.86,Z 226.132,A -85,B 0,C 180,E1 -21910.73,E2 -21910.73} C_VEL
LIN {X 0,Y 193.55,Z 224.425,A -85,B 0,C 180,E1 -21913.619,E2 -21913.619} C_VEL
LIN {X 0,Y 193.246,Z 222.667,A -85,B 0,C 180,E1 -21916.661,E2 -21916.661} C_VEL
LIN {X 0,Y 192.886,Z 220.954,A -85,B 0,C 180,E1 -21919.916,E2 -21919.916} C_VEL
LIN {X 0,Y 192.589,Z 219.488,A -85,B 0,C 180,E1 -21923.396,E2 -21923.396} C_VEL
LIN {X 0,Y 192.597,Z 219.485,A -85,B 0,C 180,E1 -21927.059,E2 -21927.059} C_VEL
LIN {X 0,Y 192.657,Z 219.48,A -85,B 0,C 180,E1 -21931.69,E2 -21931.69} C_VEL
LIN {X 0,Y 192.697,Z 219.474,A -85,B 0,C 180,E1 -21936.347,E2 -21936.347} C_VEL
LIN {X 0,Y 192.723,Z 219.473,A -85,B 0,C 180,E1 -21941.456,E2 -21941.456} C_VEL
LIN {X 0,Y 192.754,Z 219.458,A -85,B 0,C 180,E1 -21945.213,E2 -21945.213} C_VEL
LIN {X 0,Y 192.935,Z 219.435,A -85,B 0,C 180,E1 -21949.566,E2 -21949.566} C_VEL
LIN {X 0,Y 193.031,Z 219.431,A -85,B 0,C 180,E1 -21951.626,E2 -21951.626} C_VEL
LIN {X 0,Y 193.253,Z 219.411,A -85,B 0,C 180,E1 -21957.916,E2 -21957.916} C_VEL
LIN {X 0,Y 193.433,Z 219.373,A -85,B 0,C 180,E1 -21960,E2 -21960} C_VEL
LIN {X 0,Y 192.964,Z 219.435,A -85,B 0,C 180,E1 -21964.177,E2 -21964.177} C_VEL
LIN {X 0,Y 193.058,Z 219.427,A -85,B 0,C 180,E1 -21968.373,E2 -21968.373} C_VEL
LIN {X 0,Y 192.792,Z 219.461,A -85,B 0,C 180,E1 -21972.634,E2 -21972.634} C_VEL
LIN {X 0,Y 192.696,Z 219.562,A -85,B 0,C 180,E1 -21977.381,E2 -21977.381} C_VEL
LIN {X 0,Y 193.635,Z 223.704,A -85,B 0,C 180,E1 -21983.531,E2 -21983.531} C_VEL
LIN {X 0,Y 194.512,Z 227.347,A -85,B 0,C 180,E1 -21988.015,E2 -21988.015} C_VEL
LIN {X 0,Y 195.616,Z 231.531,A -85,B 0,C 180,E1 -21992.61,E2 -21992.61} C_VEL
LIN {X 0,Y 196.499,Z 235.275,A -85,B 0,C 180,E1 -21996.167,E2 -21996.167} C_VEL
LIN {X 0,Y 197.62,Z 240.642,A -85,B 0,C 180,E1 -22000.807,E2 -22000.807} C_VEL
LIN {X 0,Y 198.708,Z 246.054,A -85,B 0,C 180,E1 -22005.021,E2 -22005.021} C_VEL
LIN {X 0,Y 199.947,Z 251.704,A -85,B 0,C 180,E1 -22009.113,E2 -22009.113} C_VEL
LIN {X 0,Y 201.17,Z 258.302,A -85,B 0,C 180,E1 -22013.569,E2 -22013.569} C_VEL
LIN {X 0,Y 199.702,Z 262.03,A -85,B 0,C 180,E1 -22015.735,E2 -22015.735} C_VEL
LIN {X 0,Y 198.547,Z 264.72,A -85,B 0,C 180,E1 -22017.282,E2 -22017.282} C_VEL
LIN {X 0,Y 199.743,Z 277.657,A -85,B 0,C 180,E1 -22018.477,E2 -22018.477} C_VEL
LIN {X 0,Y 199.985,Z 289.053,A -85,B 0,C 180,E1 -22019.817,E2 -22019.817} C_VEL
LIN {X 0,Y 199.696,Z 300.204,A -85,B 0,C 180,E1 -22021.481,E2 -22021.481} C_VEL
LIN {X 0,Y 198.765,Z 309.709,A -85,B 0,C 180,E1 -22023.207,E2 -22023.207} C_VEL
LIN {X 0,Y 197.945,Z 318.126,A -85,B 0,C 180,E1 -22025.066,E2 -22025.066} C_VEL
LIN {X 0,Y 197.16,Z 325.241,A -85,B 0,C 180,E1 -22026.917,E2 -22026.917} C_VEL
LIN {X 0,Y 195.291,Z 333.087,A -85,B 0,C 180,E1 -22029.314,E2 -22029.314} C_VEL
LIN {X 0,Y 193.652,Z 340.364,A -85,B 0,C 180,E1 -22032.035,E2 -22032.035} C_VEL
LIN {X 0,Y 192.481,Z 346.92,A -85,B 0,C 180,E1 -22035.194,E2 -22035.194} C_VEL
LIN {X 0,Y 192.146,Z 349.77,A -85,B 0,C 180,E1 -22036.869,E2 -22036.869} C_VEL
LIN {X 0,Y 191.363,Z 351.416,A -85,B 0,C 180,E1 -22037.951,E2 -22037.951} C_VEL
LIN {X 0,Y 188.468,Z 353.541,A -85,B 0,C 180,E1 -22039.705,E2 -22039.705} C_VEL
LIN {X 0,Y 185.68,Z 355.697,A -85,B 0,C 180,E1 -22041.449,E2 -22041.449} C_VEL
LIN {X 0,Y 185.031,Z 357.678,A -85,B 0,C 180,E1 -22042.478,E2 -22042.478} C_VEL
LIN {X 0,Y 185.011,Z 364.56,A -85,B 0,C 180,E1 -22045.646,E2 -22045.646} C_VEL
LIN {X 0,Y 185.089,Z 370.205,A -85,B 0,C 180,E1 -22048.915,E2 -22048.915} C_VEL
LIN {X 0,Y 184.97,Z 373.207,A -85,B 0,C 180,E1 -22051.091,E2 -22051.091} C_VEL
LIN {X 0,Y 184.255,Z 376.66,A -85,B 0,C 180,E1 -22054.378,E2 -22054.378} C_VEL
LIN {X 0,Y 184.063,Z 379.903,A -85,B 0,C 180,E1 -22058.788,E2 -22058.788} C_VEL
LIN {X 0,Y 184.946,Z 381.812,A -85,B 0,C 180,E1 -22063.182,E2 -22063.182} C_VEL
LIN {X 0,Y 187.081,Z 382.505,A -85,B 0,C 180,E1 -22067.492,E2 -22067.492} C_VEL
LIN {X 0,Y 190.666,Z 382.025,A -85,B 0,C 180,E1 -22071.632,E2 -22071.632} C_VEL
LIN {X 0,Y 195.362,Z 380.361,A -85,B 0,C 180,E1 -22075.578,E2 -22075.578} C_VEL
LIN {X 0,Y 201.202,Z 377.539,A -85,B 0,C 180,E1 -22079.279,E2 -22079.279} C_VEL
LIN {X 0,Y 208.41,Z 373.485,A -85,B 0,C 180,E1 -22082.656,E2 -22082.656} C_VEL
LIN {X 0,Y 216.652,Z 368.137,A -85,B 0,C 180,E1 -22085.728,E2 -22085.728} C_VEL
LIN {X 0,Y 225.759,Z 361.43,A -85,B 0,C 180,E1 -22088.51,E2 -22088.51} C_VEL
LIN {X 0,Y 235.529,Z 353.254,A -85,B 0,C 180,E1 -22091.033,E2 -22091.033} C_VEL
LIN {X 0,Y 242.417,Z 346.741,A -85,B 0,C 180,E1 -22092.823,E2 -22092.823} C_VEL
LIN {X 0,Y 246.747,Z 342.247,A -85,B 0,C 180,E1 -22094.127,E2 -22094.127} C_VEL
LIN {X 0,Y 247.733,Z 341.005,A -85,B 0,C 180,E1 -22094.827,E2 -22094.827} C_VEL
LIN {X 0,Y 246.371,Z 341.693,A -85,B 0,C 180,E1 -22096.794,E2 -22096.794} C_VEL
LIN {X 0,Y 243.012,Z 344.545,A -85,B 0,C 180,E1 -22099.103,E2 -22099.103} C_VEL
LIN {X 0,Y 241.327,Z 346.045,A -85,B 0,C 180,E1 -22100.157,E2 -22100.157} C_VEL
LIN {X 0,Y 239.13,Z 347.904,A -85,B 0,C 180,E1 -22100.811,E2 -22100.811} C_VEL
LIN {X 0,Y 231.821,Z 353.493,A -85,B 0,C 180,E1 -22102.675,E2 -22102.675} C_VEL
LIN {X 0,Y 222.723,Z 359.5,A -85,B 0,C 180,E1 -22105.39,E2 -22105.39} C_VEL
LIN {X 0,Y 214.341,Z 364.125,A -85,B 0,C 180,E1 -22108.357,E2 -22108.357} C_VEL
LIN {X 0,Y 206.868,Z 367.322,A -85,B 0,C 180,E1 -22111.6,E2 -22111.6} C_VEL
LIN {X 0,Y 200.368,Z 369.246,A -85,B 0,C 180,E1 -22115.108,E2 -22115.108} C_VEL
LIN {X 0,Y 194.986,Z 369.925,A -85,B 0,C 180,E1 -22118.873,E2 -22118.873} C_VEL
LIN {X 0,Y 190.572,Z 369.357,A -85,B 0,C 180,E1 -22122.841,E2 -22122.841} C_VEL
LIN {X 0,Y 188.867,Z 368.573,A -85,B 0,C 180,E1 -22124.901,E2 -22124.901} C_VEL
LIN {X 0,Y 187.168,Z 367.469,A -85,B 0,C 180,E1 -22126.98,E2 -22126.98} C_VEL
LIN {X 0,Y 185.081,Z 364.284,A -85,B 0,C 180,E1 -22131.264,E2 -22131.264} C_VEL
LIN {X 0,Y 184.272,Z 360.995,A -85,B 0,C 180,E1 -22134.529,E2 -22134.529} C_VEL
LIN {X 0,Y 183.625,Z 355.233,A -85,B 0,C 180,E1 -22138.904,E2 -22138.904} C_VEL
LIN {X 0,Y 183.701,Z 348.682,A -85,B 0,C 180,E1 -22142.741,E2 -22142.741} C_VEL
LIN {X 0,Y 183.993,Z 340.44,A -85,B 0,C 180,E1 -22146.58,E2 -22146.58} C_VEL
LIN {X 0,Y 184.634,Z 331.769,A -85,B 0,C 180,E1 -22149.863,E2 -22149.863} C_VEL
LIN {X 0,Y 185.578,Z 321.132,A -85,B 0,C 180,E1 -22153.134,E2 -22153.134} C_VEL
LIN {X 0,Y 186.863,Z 309.235,A -85,B 0,C 180,E1 -22156.104,E2 -22156.104} C_VEL
LIN {X 0,Y 188.116,Z 297.252,A -85,B 0,C 180,E1 -22158.516,E2 -22158.516} C_VEL
LIN {X 0,Y 189.158,Z 286.805,A -85,B 0,C 180,E1 -22160.227,E2 -22160.227} C_VEL
LIN {X 0,Y 187.358,Z 273.208,A -85,B 0,C 180,E1 -22162.031,E2 -22162.031} C_VEL
LIN {X 0,Y 185.85,Z 258.717,A -85,B 0,C 180,E1 -22163.506,E2 -22163.506} C_VEL
LIN {X 0,Y 185.823,Z 257.217,A -85,B 0,C 180,E1 -22163.694,E2 -22163.694} C_VEL
LIN {X 0,Y 186.637,Z 247.861,A -85,B 0,C 180,E1 -22169.31,E2 -22169.31} C_VEL
LIN {X 0,Y 187.586,Z 239.293,A -85,B 0,C 180,E1 -22174.484,E2 -22174.484} C_VEL
LIN {X 0,Y 187.966,Z 234.395,A -85,B 0,C 180,E1 -22177.476,E2 -22177.476} C_VEL
LIN {X 0,Y 187.154,Z 228.377,A -85,B 0,C 180,E1 -22181.316,E2 -22181.316} C_VEL
LIN {X 0,Y 186.442,Z 224.765,A -85,B 0,C 180,E1 -22183.729,E2 -22183.729} C_VEL
LIN {X 0,Y 186.792,Z 226.806,A -85,B 0,C 180,E1 -22187.368,E2 -22187.368} C_VEL
LIN {X 0,Y 187.276,Z 229.626,A -85,B 0,C 180,E1 -22192.007,E2 -22192.007} C_VEL
LIN {X 0,Y 187.614,Z 232.207,A -85,B 0,C 180,E1 -22195.81,E2 -22195.81} C_VEL
LIN {X 0,Y 187.665,Z 235.895,A -85,B 0,C 180,E1 -22200.689,E2 -22200.689} C_VEL
LIN {X 0,Y 187.68,Z 236.084,A -85,B 0,C 180,E1 -22200.839,E2 -22200.839} C_VEL
LIN {X 0,Y 191.397,Z 245.59,A -85,B 0,C 180,E1 -22202.381,E2 -22202.381} C_VEL
LIN {X 0,Y 194.363,Z 254.951,A -85,B 0,C 180,E1 -22204.113,E2 -22204.113} C_VEL
LIN {X 0,Y 195.993,Z 262.491,A -85,B 0,C 180,E1 -22205.679,E2 -22205.679} C_VEL
LIN {X 0,Y 197.042,Z 269.795,A -85,B 0,C 180,E1 -22207.378,E2 -22207.378} C_VEL
LIN {X 0,Y 197.346,Z 273.034,A -85,B 0,C 180,E1 -22208.183,E2 -22208.183} C_VEL
LIN {X 0,Y 195.643,Z 280.476,A -85,B 0,C 180,E1 -22210.043,E2 -22210.043} C_VEL
LIN {X 0,Y 193.297,Z 288.342,A -85,B 0,C 180,E1 -22212.542,E2 -22212.542} C_VEL
LIN {X 0,Y 191.197,Z 294.363,A -85,B 0,C 180,E1 -22215.087,E2 -22215.087} C_VEL
LIN {X 0,Y 189.799,Z 298.175,A -85,B 0,C 180,E1 -22217.161,E2 -22217.161} C_VEL
LIN {X 0,Y 188.617,Z 302.453,A -85,B 0,C 180,E1 -22220.345,E2 -22220.345} C_VEL
LIN {X 0,Y 187.27,Z 305.416,A -85,B 0,C 180,E1 -22223.533,E2 -22223.533} C_VEL
LIN {X 0,Y 186.864,Z 306.649,A -85,B 0,C 180,E1 -22225.683,E2 -22225.683} C_VEL
LIN {X 0,Y 186.52,Z 307.407,A -85,B 0,C 180,E1 -22227.838,E2 -22227.838} C_VEL
LIN {X 0,Y 186.391,Z 307.681,A -85,B 0,C 180,E1 -22229.997,E2 -22229.997} C_VEL
LIN {X 0,Y 186.519,Z 307.44,A -85,B 0,C 180,E1 -22232.157,E2 -22232.157} C_VEL
LIN {X 0,Y 186.862,Z 306.727,A -85,B 0,C 180,E1 -22234.311,E2 -22234.311} C_VEL
LIN {X 0,Y 187.267,Z 305.533,A -85,B 0,C 180,E1 -22236.462,E2 -22236.462} C_VEL
LIN {X 0,Y 188.602,Z 302.625,A -85,B 0,C 180,E1 -22239.65,E2 -22239.65} C_VEL
LIN {X 0,Y 189.755,Z 298.432,A -85,B 0,C 180,E1 -22242.837,E2 -22242.837} C_VEL
LIN {X 0,Y 190.639,Z 296.627,A -85,B 0,C 180,E1 -22243.862,E2 -22243.862} C_VEL
LIN {X 0,Y 191.921,Z 292.492,A -85,B 0,C 180,E1 -22245.938,E2 -22245.938} C_VEL
LIN {X 0,Y 194.212,Z 285.887,A -85,B 0,C 180,E1 -22248.457,E2 -22248.457} C_VEL
LIN {X 0,Y 196.261,Z 278.227,A -85,B 0,C 180,E1 -22250.706,E2 -22250.706} C_VEL
LIN {X 0,Y 197.372,Z 272.04,A -85,B 0,C 180,E1 -22252.209,E2 -22252.209} C_VEL
LIN {X 0,Y 196.198,Z 263.063,A -85,B 0,C 180,E1 -22254.368,E2 -22254.368} C_VEL
LIN {X 0,Y 193.987,Z 253.569,A -85,B 0,C 180,E1 -22256.319,E2 -22256.319} C_VEL
LIN {X 0,Y 190.8,Z 243.877,A -85,B 0,C 180,E1 -22258.075,E2 -22258.075} C_VEL
LIN {X 0,Y 187.715,Z 235.975,A -85,B 0,C 180,E1 -22259.4,E2 -22259.4} C_VEL
LIN {X 0,Y 187.657,Z 232.371,A -85,B 0,C 180,E1 -22264.174,E2 -22264.174} C_VEL
LIN {X 0,Y 187.339,Z 229.775,A -85,B 0,C 180,E1 -22268.018,E2 -22268.018} C_VEL
LIN {X 0,Y 186.781,Z 226.959,A -85,B 0,C 180,E1 -22272.627,E2 -22272.627} C_VEL
LIN {X 0,Y 186.373,Z 224.402,A -85,B 0,C 180,E1 -22277.252,E2 -22277.252} C_VEL
LIN {X 0,Y 186.086,Z 223.012,A -85,B 0,C 180,E1 -22280.055,E2 -22280.055} C_VEL
LIN {X 0,Y 185.539,Z 220.649,A -85,B 0,C 180,E1 -22285.376,E2 -22285.376} C_VEL
LIN {X 0,Y 185.526,Z 220.364,A -85,B 0,C 180,E1 -22286.443,E2 -22286.443} C_VEL
LIN {X 0,Y 185.574,Z 220.356,A -85,B 0,C 180,E1 -22290.574,E2 -22290.574} C_VEL
LIN {X 0,Y 185.579,Z 220.354,A -85,B 0,C 180,E1 -22295.381,E2 -22295.381} C_VEL
LIN {X 0,Y 185.599,Z 220.35,A -85,B 0,C 180,E1 -22300.074,E2 -22300.074} C_VEL
LIN {X 0,Y 185.685,Z 220.337,A -85,B 0,C 180,E1 -22304.636,E2 -22304.636} C_VEL
LIN {X 0,Y 185.879,Z 220.314,A -85,B 0,C 180,E1 -22309.417,E2 -22309.417} C_VEL
LIN {X 0,Y 185.942,Z 220.314,A -85,B 0,C 180,E1 -22313.489,E2 -22313.489} C_VEL
LIN {X 0,Y 186.197,Z 220.29,A -85,B 0,C 180,E1 -22317.837,E2 -22317.837} C_VEL
LIN {X 0,Y 186.397,Z 220.249,A -85,B 0,C 180,E1 -22320,E2 -22320} C_VEL
LIN {X 0,Y 185.912,Z 220.313,A -85,B 0,C 180,E1 -22324.336,E2 -22324.336} C_VEL
LIN {X 0,Y 186.004,Z 220.303,A -85,B 0,C 180,E1 -22328.693,E2 -22328.693} C_VEL
LIN {X 0,Y 185.697,Z 220.342,A -85,B 0,C 180,E1 -22333.682,E2 -22333.682} C_VEL
LIN {X 0,Y 186.155,Z 222.361,A -85,B 0,C 180,E1 -22337.579,E2 -22337.579} C_VEL
LIN {X 0,Y 186.721,Z 225.26,A -85,B 0,C 180,E1 -22342.11,E2 -22342.11} C_VEL
LIN {X 0,Y 187.562,Z 228.784,A -85,B 0,C 180,E1 -22346.721,E2 -22346.721} C_VEL
LIN {X 0,Y 188.646,Z 232.83,A -85,B 0,C 180,E1 -22351.438,E2 -22351.438} C_VEL
LIN {X 0,Y 189.786,Z 237.677,A -85,B 0,C 180,E1 -22356.335,E2 -22356.335} C_VEL
LIN {X 0,Y 191.004,Z 243.532,A -85,B 0,C 180,E1 -22361.476,E2 -22361.476} C_VEL
LIN {X 0,Y 192.414,Z 250.446,A -85,B 0,C 180,E1 -22366.929,E2 -22366.929} C_VEL
LIN {X 0,Y 193.517,Z 255.833,A -85,B 0,C 180,E1 -22370.883,E2 -22370.883} C_VEL
LIN {X 0,Y 194.058,Z 258.602,A -85,B 0,C 180,E1 -22372.821,E2 -22372.821} C_VEL
LIN {X 0,Y 193.955,Z 259.933,A -85,B 0,C 180,E1 -22373.689,E2 -22373.689} C_VEL
LIN {X 0,Y 192.139,Z 264.134,A -85,B 0,C 180,E1 -22376.188,E2 -22376.188} C_VEL
LIN {X 0,Y 193.242,Z 276.562,A -85,B 0,C 180,E1 -22377.365,E2 -22377.365} C_VEL
LIN {X 0,Y 193.508,Z 288.446,A -85,B 0,C 180,E1 -22378.821,E2 -22378.821} C_VEL
LIN {X 0,Y 193.123,Z 300.18,A -85,B 0,C 180,E1 -22380.656,E2 -22380.656} C_VEL
LIN {X 0,Y 192.08,Z 309.772,A -85,B 0,C 180,E1 -22382.491,E2 -22382.491} C_VEL
LIN {X 0,Y 191.149,Z 318.04,A -85,B 0,C 180,E1 -22384.408,E2 -22384.408} C_VEL
LIN {X 0,Y 190.513,Z 324.156,A -85,B 0,C 180,E1 -22386.063,E2 -22386.063} C_VEL
LIN {X 0,Y 188.863,Z 330.957,A -85,B 0,C 180,E1 -22388.157,E2 -22388.157} C_VEL
LIN {X 0,Y 187.175,Z 338.072,A -85,B 0,C 180,E1 -22390.823,E2 -22390.823} C_VEL
LIN {X 0,Y 185.879,Z 343.89,A -85,B 0,C 180,E1 -22393.53,E2 -22393.53} C_VEL
LIN {X 0,Y 185.066,Z 349.494,A -85,B 0,C 180,E1 -22396.832,E2 -22396.832} C_VEL
LIN {X 0,Y 184.933,Z 353.881,A -85,B 0,C 180,E1 -22400.267,E2 -22400.267} C_VEL
LIN {X 0,Y 185.066,Z 355.336,A -85,B 0,C 180,E1 -22401.525,E2 -22401.525} C_VEL
LIN {X 0,Y 185.031,Z 357.678,A -85,B 0,C 180,E1 -22402.478,E2 -22402.478} C_VEL
LIN {X 0,Y 184.454,Z 361,A -85,B 0,C 180,E1 -22403.979,E2 -22403.979} C_VEL
LIN {X 0,Y 183.027,Z 363.853,A -85,B 0,C 180,E1 -22405.541,E2 -22405.541} C_VEL
LIN {X 0,Y 179.488,Z 368.577,A -85,B 0,C 180,E1 -22408.861,E2 -22408.861} C_VEL
LIN {X 0,Y 178.09,Z 371.453,A -85,B 0,C 180,E1 -22411.228,E2 -22411.228} C_VEL
LIN {X 0,Y 177.372,Z 375.009,A -85,B 0,C 180,E1 -22414.548,E2 -22414.548} C_VEL
LIN {X 0,Y 177.172,Z 378.559,A -85,B 0,C 180,E1 -22419.133,E2 -22419.133} C_VEL
LIN {X 0,Y 178.085,Z 380.781,A -85,B 0,C 180,E1 -22423.7,E2 -22423.7} C_VEL
LIN {X 0,Y 180.332,Z 381.806,A -85,B 0,C 180,E1 -22428.169,E2 -22428.169} C_VEL
LIN {X 0,Y 184.08,Z 381.68,A -85,B 0,C 180,E1 -22432.447,E2 -22432.447} C_VEL
LIN {X 0,Y 188.98,Z 380.386,A -85,B 0,C 180,E1 -22436.507,E2 -22436.507} C_VEL
LIN {X 0,Y 195.061,Z 377.962,A -85,B 0,C 180,E1 -22440.295,E2 -22440.295} C_VEL
LIN {X 0,Y 202.527,Z 374.374,A -85,B 0,C 180,E1 -22443.729,E2 -22443.729} C_VEL
LIN {X 0,Y 211.01,Z 369.568,A -85,B 0,C 180,E1 -22446.838,E2 -22446.838} C_VEL
LIN {X 0,Y 220.378,Z 363.457,A -85,B 0,C 180,E1 -22449.631,E2 -22449.631} C_VEL
LIN {X 0,Y 231.722,Z 354.907,A -85,B 0,C 180,E1 -22452.444,E2 -22452.444} C_VEL
LIN {X 0,Y 239.103,Z 348.557,A -85,B 0,C 180,E1 -22454.276,E2 -22454.276} C_VEL
LIN {X 0,Y 241.579,Z 346.306,A -85,B 0,C 180,E1 -22454.97,E2 -22454.97} C_VEL
LIN {X 0,Y 241.674,Z 345.953,A -85,B 0,C 180,E1 -22455.738,E2 -22455.738} C_VEL
LIN {X 0,Y 239.345,Z 347.462,A -85,B 0,C 180,E1 -22457.518,E2 -22457.518} C_VEL
LIN {X 0,Y 236.505,Z 349.591,A -85,B 0,C 180,E1 -22459.175,E2 -22459.175} C_VEL
LIN {X 0,Y 226.584,Z 356.477,A -85,B 0,C 180,E1 -22461.659,E2 -22461.659} C_VEL
LIN {X 0,Y 217.172,Z 361.914,A -85,B 0,C 180,E1 -22464.373,E2 -22464.373} C_VEL
LIN {X 0,Y 208.517,Z 365.995,A -85,B 0,C 180,E1 -22467.366,E2 -22467.366} C_VEL
LIN {X 0,Y 200.775,Z 368.756,A -85,B 0,C 180,E1 -22470.655,E2 -22470.655} C_VEL
LIN {X 0,Y 194.035,Z 370.233,A -85,B 0,C 180,E1 -22474.237,E2 -22474.237} C_VEL
LIN {X 0,Y 188.408,Z 370.495,A -85,B 0,C 180,E1 -22478.098,E2 -22478.098} C_VEL
LIN {X 0,Y 183.808,Z 369.531,A -85,B 0,C 180,E1 -22482.189,E2 -22482.189} C_VEL
LIN {X 0,Y 180.285,Z 367.316,A -85,B 0,C 180,E1 -22486.473,E2 -22486.473} C_VEL
LIN {X 0,Y 178.097,Z 363.768,A -85,B 0,C 180,E1 -22490.918,E2 -22490.918} C_VEL
LIN {X 0,Y 177.247,Z 360.237,A -85,B 0,C 180,E1 -22494.311,E2 -22494.311} C_VEL
LIN {X 0,Y 176.613,Z 354.068,A -85,B 0,C 180,E1 -22498.86,E2 -22498.86} C_VEL
LIN {X 0,Y 176.718,Z 347.221,A -85,B 0,C 180,E1 -22502.85,E2 -22502.85} C_VEL
LIN {X 0,Y 177.056,Z 338.544,A -85,B 0,C 180,E1 -22506.839,E2 -22506.839} C_VEL
LIN {X 0,Y 177.748,Z 329.445,A -85,B 0,C 180,E1 -22510.249,E2 -22510.249} C_VEL
LIN {X 0,Y 178.633,Z 319.292,A -85,B 0,C 180,E1 -22513.364,E2 -22513.364} C_VEL
LIN {X 0,Y 179.826,Z 308.194,A -85,B 0,C 180,E1 -22516.169,E2 -22516.169} C_VEL
LIN {X 0,Y 181.093,Z 295.917,A -85,B 0,C 180,E1 -22518.674,E2 -22518.674} C_VEL
LIN {X 0,Y 181.98,Z 285.966,A -85,B 0,C 180,E1 -22520.339,E2 -22520.339} C_VEL
LIN {X 0,Y 180.135,Z 272.286,A -85,B 0,C 180,E1 -22522.194,E2 -22522.194} C_VEL
LIN {X 0,Y 178.73,Z 258.174,A -85,B 0,C 180,E1 -22523.654,E2 -22523.654} C_VEL
LIN {X 0,Y 178.721,Z 257.578,A -85,B 0,C 180,E1 -22523.77,E2 -22523.77} C_VEL
LIN {X 0,Y 179.559,Z 248.618,A -85,B 0,C 180,E1 -22529.292,E2 -22529.292} C_VEL
LIN {X 0,Y 180.433,Z 240.803,A -85,B 0,C 180,E1 -22534.138,E2 -22534.138} C_VEL
LIN {X 0,Y 180.924,Z 235.068,A -85,B 0,C 180,E1 -22537.721,E2 -22537.721} C_VEL
LIN {X 0,Y 180.071,Z 229.19,A -85,B 0,C 180,E1 -22541.567,E2 -22541.567} C_VEL
LIN {X 0,Y 179.58,Z 226.64,A -85,B 0,C 180,E1 -22543.356,E2 -22543.356} C_VEL
LIN {X 0,Y 179.862,Z 227.624,A -85,B 0,C 180,E1 -22545.301,E2 -22545.301} C_VEL
LIN {X 0,Y 180.073,Z 229.41,A -85,B 0,C 180,E1 -22548.43,E2 -22548.43} C_VEL
LIN {X 0,Y 180.355,Z 231.199,A -85,B 0,C 180,E1 -22551.426,E2 -22551.426} C_VEL
LIN {X 0,Y 180.633,Z 233.37,A -85,B 0,C 180,E1 -22554.792,E2 -22554.792} C_VEL
LIN {X 0,Y 180.851,Z 236.864,A -85,B 0,C 180,E1 -22559.49,E2 -22559.49} C_VEL
LIN {X 0,Y 184.959,Z 247.066,A -85,B 0,C 180,E1 -22561.302,E2 -22561.302} C_VEL
LIN {X 0,Y 187.992,Z 256.678,A -85,B 0,C 180,E1 -22563.212,E2 -22563.212} C_VEL
LIN {X 0,Y 189.734,Z 265.251,A -85,B 0,C 180,E1 -22565.127,E2 -22565.127} C_VEL
LIN {X 0,Y 190.695,Z 273.195,A -85,B 0,C 180,E1 -22567.128,E2 -22567.128} C_VEL
LIN {X 0,Y 190.443,Z 275.917,A -85,B 0,C 180,E1 -22567.836,E2 -22567.836} C_VEL
LIN {X 0,Y 188.572,Z 283.203,A -85,B 0,C 180,E1 -22569.831,E2 -22569.831} C_VEL
LIN {X 0,Y 186.611,Z 289.36,A -85,B 0,C 180,E1 -22571.896,E2 -22571.896} C_VEL
LIN {X 0,Y 184.415,Z 295.363,A -85,B 0,C 180,E1 -22574.525,E2 -22574.525} C_VEL
LIN {X 0,Y 182.951,Z 299.163,A -85,B 0,C 180,E1 -22576.671,E2 -22576.671} C_VEL
LIN {X 0,Y 181.692,Z 303.431,A -85,B 0,C 180,E1 -22579.973,E2 -22579.973} C_VEL
LIN {X 0,Y 180.289,Z 306.392,A -85,B 0,C 180,E1 -22583.281,E2 -22583.281} C_VEL
LIN {X 0,Y 179.857,Z 307.623,A -85,B 0,C 180,E1 -22585.515,E2 -22585.515} C_VEL
LIN {X 0,Y 179.498,Z 308.381,A -85,B 0,C 180,E1 -22587.753,E2 -22587.753} C_VEL
LIN {X 0,Y 179.363,Z 308.655,A -85,B 0,C 180,E1 -22589.997,E2 -22589.997} C_VEL
LIN {X 0,Y 179.497,Z 308.414,A -85,B 0,C 180,E1 -22592.241,E2 -22592.241} C_VEL
LIN {X 0,Y 179.855,Z 307.7,A -85,B 0,C 180,E1 -22594.479,E2 -22594.479} C_VEL
LIN {X 0,Y 180.286,Z 306.507,A -85,B 0,C 180,E1 -22596.713,E2 -22596.713} C_VEL
LIN {X 0,Y 181.677,Z 303.601,A -85,B 0,C 180,E1 -22600.022,E2 -22600.022} C_VEL
LIN {X 0,Y 182.907,Z 299.418,A -85,B 0,C 180,E1 -22603.326,E2 -22603.326} C_VEL
LIN {X 0,Y 183.822,Z 297.617,A -85,B 0,C 180,E1 -22604.386,E2 -22604.386} C_VEL
LIN {X 0,Y 185.175,Z 293.497,A -85,B 0,C 180,E1 -22606.535,E2 -22606.535} C_VEL
LIN {X 0,Y 187.568,Z 286.908,A -85,B 0,C 180,E1 -22609.135,E2 -22609.135} C_VEL
LIN {X 0,Y 189.482,Z 280.298,A -85,B 0,C 180,E1 -22611.197,E2 -22611.197} C_VEL
LIN {X 0,Y 190.759,Z 274.827,A -85,B 0,C 180,E1 -22612.596,E2 -22612.596} C_VEL
LIN {X 0,Y 190.118,Z 267.134,A -85,B 0,C 180,E1 -22614.594,E2 -22614.594} C_VEL
LIN {X 0,Y 188.174,Z 257.382,A -85,B 0,C 180,E1 -22616.809,E2 -22616.809} C_VEL
LIN {X 0,Y 185.496,Z 248.41,A -85,B 0,C 180,E1 -22618.605,E2 -22618.605} C_VEL
LIN {X 0,Y 181.746,Z 239.133,A -85,B 0,C 180,E1 -22620.321,E2 -22620.321} C_VEL
LIN {X 0,Y 180.837,Z 236.704,A -85,B 0,C 180,E1 -22620.739,E2 -22620.739} C_VEL
LIN {X 0,Y 180.66,Z 233.223,A -85,B 0,C 180,E1 -22625.695,E2 -22625.695} C_VEL
LIN {X 0,Y 180.382,Z 231.209,A -85,B 0,C 180,E1 -22628.809,E2 -22628.809} C_VEL
LIN {X 0,Y 180.037,Z 229.267,A -85,B 0,C 180,E1 -22632.124,E2 -22632.124} C_VEL
LIN {X 0,Y 179.723,Z 227.513,A -85,B 0,C 180,E1 -22635.26,E2 -22635.26} C_VEL
LIN {X 0,Y 179.466,Z 226.001,A -85,B 0,C 180,E1 -22638.261,E2 -22638.261} C_VEL
LIN {X 0,Y 179.122,Z 224.429,A -85,B 0,C 180,E1 -22641.689,E2 -22641.689} C_VEL
LIN {X 0,Y 178.729,Z 222.392,A -85,B 0,C 180,E1 -22646.598,E2 -22646.598} C_VEL
LIN {X 0,Y 178.515,Z 221.236,A -85,B 0,C 180,E1 -22650.005,E2 -22650.005} C_VEL
LIN {X 0,Y 178.526,Z 221.232,A -85,B 0,C 180,E1 -22654.874,E2 -22654.874} C_VEL
LIN {X 0,Y 178.615,Z 221.223,A -85,B 0,C 180,E1 -22660.782,E2 -22660.782} C_VEL
LIN {X 0,Y 178.648,Z 221.221,A -85,B 0,C 180,E1 -22666.347,E2 -22666.347} C_VEL
LIN {X 0,Y 178.905,Z 221.184,A -85,B 0,C 180,E1 -22670.959,E2 -22670.959} C_VEL
LIN {X 0,Y 178.858,Z 221.187,A -85,B 0,C 180,E1 -22675.492,E2 -22675.492} C_VEL
LIN {X 0,Y 179.36,Z 221.125,A -85,B 0,C 180,E1 -22680,E2 -22680} C_VEL
LIN {X 0,Y 178.86,Z 221.19,A -85,B 0,C 180,E1 -22684.507,E2 -22684.507} C_VEL
LIN {X 0,Y 178.954,Z 221.18,A -85,B 0,C 180,E1 -22689.038,E2 -22689.038} C_VEL
LIN {X 0,Y 178.915,Z 221.645,A -85,B 0,C 180,E1 -22690.897,E2 -22690.897} C_VEL
LIN {X 0,Y 179.274,Z 224.098,A -85,B 0,C 180,E1 -22695.927,E2 -22695.927} C_VEL
LIN {X 0,Y 179.833,Z 226.713,A -85,B 0,C 180,E1 -22700.302,E2 -22700.302} C_VEL
LIN {X 0,Y 180.678,Z 230.113,A -85,B 0,C 180,E1 -22705.333,E2 -22705.333} C_VEL
LIN {X 0,Y 181.661,Z 234.097,A -85,B 0,C 180,E1 -22710.195,E2 -22710.195} C_VEL
LIN {X 0,Y 182.834,Z 238.748,A -85,B 0,C 180,E1 -22715.211,E2 -22715.211} C_VEL
LIN {X 0,Y 183.955,Z 244.433,A -85,B 0,C 180,E1 -22720.503,E2 -22720.503} C_VEL
LIN {X 0,Y 185.301,Z 251.132,A -85,B 0,C 180,E1 -22726.106,E2 -22726.106} C_VEL
LIN {X 0,Y 186.398,Z 256.391,A -85,B 0,C 180,E1 -22730.14,E2 -22730.14} C_VEL
LIN {X 0,Y 187.039,Z 260.396,A -85,B 0,C 180,E1 -22733.048,E2 -22733.048} C_VEL
LIN {X 0,Y 185.812,Z 263.355,A -85,B 0,C 180,E1 -22734.944,E2 -22734.944} C_VEL
LIN {X 0,Y 186.964,Z 277.742,A -85,B 0,C 180,E1 -22736.445,E2 -22736.445} C_VEL
LIN {X 0,Y 187.051,Z 288.902,A -85,B 0,C 180,E1 -22737.907,E2 -22737.907} C_VEL
LIN {X 0,Y 186.562,Z 300.138,A -85,B 0,C 180,E1 -22739.765,E2 -22739.765} C_VEL
LIN {X 0,Y 185.432,Z 309.837,A -85,B 0,C 180,E1 -22741.725,E2 -22741.725} C_VEL
LIN {X 0,Y 184.391,Z 317.957,A -85,B 0,C 180,E1 -22743.703,E2 -22743.703} C_VEL
LIN {X 0,Y 183.529,Z 324.838,A -85,B 0,C 180,E1 -22745.694,E2 -22745.694} C_VEL
LIN {X 0,Y 181.844,Z 331.248,A -85,B 0,C 180,E1 -22747.809,E2 -22747.809} C_VEL
LIN {X 0,Y 180.085,Z 338.321,A -85,B 0,C 180,E1 -22750.63,E2 -22750.63} C_VEL
LIN {X 0,Y 178.574,Z 344.889,A -85,B 0,C 180,E1 -22754.012,E2 -22754.012} C_VEL
LIN {X 0,Y 177.913,Z 350.064,A -85,B 0,C 180,E1 -22757.455,E2 -22757.455} C_VEL
LIN {X 0,Y 177.908,Z 353.969,A -85,B 0,C 180,E1 -22760.964,E2 -22760.964} C_VEL
LIN {X 0,Y 178.112,Z 355.431,A -85,B 0,C 180,E1 -22762.37,E2 -22762.37} C_VEL
LIN {X 0,Y 178.148,Z 362.217,A -85,B 0,C 180,E1 -22765.478,E2 -22765.478} C_VEL
LIN {X 0,Y 178.213,Z 368.162,A -85,B 0,C 180,E1 -22768.873,E2 -22768.873} C_VEL
LIN {X 0,Y 178.09,Z 371.453,A -85,B 0,C 180,E1 -22771.228,E2 -22771.228} C_VEL
LIN {X 0,Y 177.525,Z 372.767,A -85,B 0,C 180,E1 -22772.411,E2 -22772.411} C_VEL
LIN {X 0,Y 175.213,Z 374.676,A -85,B 0,C 180,E1 -22774.787,E2 -22774.787} C_VEL
LIN {X 0,Y 171.35,Z 376.692,A -85,B 0,C 180,E1 -22778.481,E2 -22778.481} C_VEL
LIN {X 0,Y 170.462,Z 377.702,A -85,B 0,C 180,E1 -22780.429,E2 -22780.429} C_VEL
LIN {X 0,Y 170.468,Z 378.056,A -85,B 0,C 180,E1 -22781.085,E2 -22781.085} C_VEL
LIN {X 0,Y 171.245,Z 379.622,A -85,B 0,C 180,E1 -22784.258,E2 -22784.258} C_VEL
LIN {X 0,Y 173.627,Z 380.954,A -85,B 0,C 180,E1 -22788.897,E2 -22788.897} C_VEL
LIN {X 0,Y 177.54,Z 381.176,A -85,B 0,C 180,E1 -22793.322,E2 -22793.322} C_VEL
LIN {X 0,Y 182.653,Z 380.274,A -85,B 0,C 180,E1 -22797.502,E2 -22797.502} C_VEL
LIN {X 0,Y 188.973,Z 378.273,A -85,B 0,C 180,E1 -22801.38,E2 -22801.38} C_VEL
LIN {X 0,Y 196.695,Z 375.148,A -85,B 0,C 180,E1 -22804.871,E2 -22804.871} C_VEL
LIN {X 0,Y 206.712,Z 370.2,A -85,B 0,C 180,E1 -22808.407,E2 -22808.407} C_VEL
LIN {X 0,Y 215.066,Z 365.338,A -85,B 0,C 180,E1 -22810.814,E2 -22810.814} C_VEL
LIN {X 0,Y 225.435,Z 358.445,A -85,B 0,C 180,E1 -22813.306,E2 -22813.306} C_VEL
LIN {X 0,Y 234.464,Z 351.608,A -85,B 0,C 180,E1 -22815.392,E2 -22815.392} C_VEL
LIN {X 0,Y 235.683,Z 350.61,A -85,B 0,C 180,E1 -22815.701,E2 -22815.701} C_VEL
LIN {X 0,Y 234.757,Z 351.095,A -85,B 0,C 180,E1 -22816.484,E2 -22816.484} C_VEL
LIN {X 0,Y 231.647,Z 353.038,A -85,B 0,C 180,E1 -22818.128,E2 -22818.128} C_VEL
LIN {X 0,Y 221.378,Z 359.317,A -85,B 0,C 180,E1 -22820.585,E2 -22820.585} C_VEL
LIN {X 0,Y 211.674,Z 364.206,A -85,B 0,C 180,E1 -22823.299,E2 -22823.299} C_VEL
LIN {X 0,Y 202.528,Z 367.825,A -85,B 0,C 180,E1 -22826.395,E2 -22826.395} C_VEL
LIN {X 0,Y 194.718,Z 370.042,A -85,B 0,C 180,E1 -22829.648,E2 -22829.648} C_VEL
LIN {X 0,Y 187.728,Z 371.119,A -85,B 0,C 180,E1 -22833.305,E2 -22833.305} C_VEL
LIN {X 0,Y 181.876,Z 370.964,A -85,B 0,C 180,E1 -22837.268,E2 -22837.268} C_VEL
LIN {X 0,Y 177.085,Z 369.594,A -85,B 0,C 180,E1 -22841.488,E2 -22841.488} C_VEL
LIN {X 0,Y 173.414,Z 366.994,A -85,B 0,C 180,E1 -22845.927,E2 -22845.927} C_VEL
LIN {X 0,Y 171.133,Z 363.132,A -85,B 0,C 180,E1 -22850.545,E2 -22850.545} C_VEL
LIN {X 0,Y 170.254,Z 359.3,A -85,B 0,C 180,E1 -22854.077,E2 -22854.077} C_VEL
LIN {X 0,Y 169.704,Z 354.572,A -85,B 0,C 180,E1 -22857.627,E2 -22857.627} C_VEL
LIN {X 0,Y 169.691,Z 347.805,A -85,B 0,C 180,E1 -22861.78,E2 -22861.78} C_VEL
LIN {X 0,Y 169.888,Z 340.625,A -85,B 0,C 180,E1 -22865.341,E2 -22865.341} C_VEL
LIN {X 0,Y 170.502,Z 331.469,A -85,B 0,C 180,E1 -22869.057,E2 -22869.057} C_VEL
LIN {X 0,Y 171.362,Z 321.361,A -85,B 0,C 180,E1 -22872.434,E2 -22872.434} C_VEL
LIN {X 0,Y 172.578,Z 309.439,A -85,B 0,C 180,E1 -22875.652,E2 -22875.652} C_VEL
LIN {X 0,Y 173.85,Z 297.537,A -85,B 0,C 180,E1 -22878.258,E2 -22878.258} C_VEL
LIN {X 0,Y 174.857,Z 286.081,A -85,B 0,C 180,E1 -22880.284,E2 -22880.284} C_VEL
LIN {X 0,Y 172.95,Z 271.854,A -85,B 0,C 180,E1 -22882.271,E2 -22882.271} C_VEL
LIN {X 0,Y 171.642,Z 257.94,A -85,B 0,C 180,E1 -22883.818,E2 -22883.818} C_VEL
LIN {X 0,Y 172.455,Z 249.326,A -85,B 0,C 180,E1 -22889.277,E2 -22889.277} C_VEL
LIN {X 0,Y 173.422,Z 241.023,A -85,B 0,C 180,E1 -22894.566,E2 -22894.566} C_VEL
LIN {X 0,Y 173.877,Z 236.715,A -85,B 0,C 180,E1 -22897.322,E2 -22897.322} C_VEL
LIN {X 0,Y 173.381,Z 232.034,A -85,B 0,C 180,E1 -22900.434,E2 -22900.434} C_VEL
LIN {X 0,Y 172.717,Z 228.551,A -85,B 0,C 180,E1 -22902.905,E2 -22902.905} C_VEL
LIN {X 0,Y 173.125,Z 230.59,A -85,B 0,C 180,E1 -22906.946,E2 -22906.946} C_VEL
LIN {X 0,Y 173.415,Z 232.515,A -85,B 0,C 180,E1 -22910.356,E2 -22910.356} C_VEL
LIN {X 0,Y 173.785,Z 235.751,A -85,B 0,C 180,E1 -22915.513,E2 -22915.513} C_VEL
LIN {X 0,Y 173.891,Z 237.468,A -85,B 0,C 180,E1 -22917.967,E2 -22917.967} C_VEL
LIN {X 0,Y 175.451,Z 240.862,A -85,B 0,C 180,E1 -22918.615,E2 -22918.615} C_VEL
LIN {X 0,Y 179.068,Z 249.909,A -85,B 0,C 180,E1 -22920.419,E2 -22920.419} C_VEL
LIN {X 0,Y 181.696,Z 258.828,A -85,B 0,C 180,E1 -22922.341,E2 -22922.341} C_VEL
LIN {X 0,Y 183.476,Z 267.954,A -85,B 0,C 180,E1 -22924.529,E2 -22924.529} C_VEL
LIN {X 0,Y 184.225,Z 275.61,A -85,B 0,C 180,E1 -22926.629,E2 -22926.629} C_VEL
LIN {X 0,Y 182.523,Z 282.581,A -85,B 0,C 180,E1 -22928.541,E2 -22928.541} C_VEL
LIN {X 0,Y 180.468,Z 288.975,A -85,B 0,C 180,E1 -22930.667,E2 -22930.667} C_VEL
LIN {X 0,Y 178.02,Z 295.295,A -85,B 0,C 180,E1 -22933.365,E2 -22933.365} C_VEL
LIN {X 0,Y 176.118,Z 300.151,A -85,B 0,C 180,E1 -22936.144,E2 -22936.144} C_VEL
LIN {X 0,Y 174.775,Z 304.408,A -85,B 0,C 180,E1 -22939.572,E2 -22939.572} C_VEL
LIN {X 0,Y 173.311,Z 307.368,A -85,B 0,C 180,E1 -22943.009,E2 -22943.009} C_VEL
LIN {X 0,Y 172.852,Z 308.596,A -85,B 0,C 180,E1 -22945.333,E2 -22945.333} C_VEL
LIN {X 0,Y 172.476,Z 309.355,A -85,B 0,C 180,E1 -22947.662,E2 -22947.662} C_VEL
LIN {X 0,Y 172.335,Z 309.629,A -85,B 0,C 180,E1 -22949.997,E2 -22949.997} C_VEL
LIN {X 0,Y 172.475,Z 309.388,A -85,B 0,C 180,E1 -22952.332,E2 -22952.332} C_VEL
LIN {X 0,Y 172.85,Z 308.674,A -85,B 0,C 180,E1 -22954.661,E2 -22954.661} C_VEL
LIN {X 0,Y 173.309,Z 307.48,A -85,B 0,C 180,E1 -22956.985,E2 -22956.985} C_VEL
LIN {X 0,Y 174.76,Z 304.579,A -85,B 0,C 180,E1 -22960.423,E2 -22960.423} C_VEL
LIN {X 0,Y 176.074,Z 300.404,A -85,B 0,C 180,E1 -22963.853,E2 -22963.853} C_VEL
LIN {X 0,Y 177.023,Z 298.609,A -85,B 0,C 180,E1 -22964.952,E2 -22964.952} C_VEL
LIN {X 0,Y 178.451,Z 294.502,A -85,B 0,C 180,E1 -22967.177,E2 -22967.177} C_VEL
LIN {X 0,Y 180.951,Z 287.926,A -85,B 0,C 180,E1 -22969.864,E2 -22969.864} C_VEL
LIN {X 0,Y 183.456,Z 279.394,A -85,B 0,C 180,E1 -22972.522,E2 -22972.522} C_VEL
LIN {X 0,Y 184.265,Z 276.111,A -85,B 0,C 180,E1 -22973.382,E2 -22973.382} C_VEL
LIN {X 0,Y 183.632,Z 268.46,A -85,B 0,C 180,E1 -22975.5,E2 -22975.5} C_VEL
LIN {X 0,Y 181.957,Z 259.783,A -85,B 0,C 180,E1 -22977.609,E2 -22977.609} C_VEL
LIN {X 0,Y 179.814,Z 252.077,A -85,B 0,C 180,E1 -22979.297,E2 -22979.297} C_VEL
LIN {X 0,Y 176.483,Z 243.223,A -85,B 0,C 180,E1 -22981.111,E2 -22981.111} C_VEL
LIN {X 0,Y 173.943,Z 237.418,A -85,B 0,C 180,E1 -22982.278,E2 -22982.278} C_VEL
LIN {X 0,Y 173.796,Z 234.923,A -85,B 0,C 180,E1 -22986.024,E2 -22986.024} C_VEL
LIN {X 0,Y 173.351,Z 232.225,A -85,B 0,C 180,E1 -22990.437,E2 -22990.437} C_VEL
LIN {X 0,Y 173.042,Z 230.439,A -85,B 0,C 180,E1 -22993.661,E2 -22993.661} C_VEL
LIN {X 0,Y 172.764,Z 228.705,A -85,B 0,C 180,E1 -22997.069,E2 -22997.069} C_VEL
LIN {X 0,Y 172.299,Z 226.383,A -85,B 0,C 180,E1 -23002.277,E2 -23002.277} C_VEL
LIN {X 0,Y 172.065,Z 225.218,A -85,B 0,C 180,E1 -23005.122,E2 -23005.122} C_VEL
LIN {X 0,Y 171.716,Z 223.326,A -85,B 0,C 180,E1 -23010.584,E2 -23010.584} C_VEL
LIN {X 0,Y 171.45,Z 222.115,A -85,B 0,C 180,E1 -23015.8,E2 -23015.8} C_VEL
LIN {X 0,Y 171.571,Z 222.1,A -85,B 0,C 180,E1 -23020.87,E2 -23020.87} C_VEL
LIN {X 0,Y 171.566,Z 222.098,A -85,B 0,C 180,E1 -23025.772,E2 -23025.772} C_VEL
LIN {X 0,Y 171.84,Z 222.061,A -85,B 0,C 180,E1 -23030.584,E2 -23030.584} C_VEL
LIN {X 0,Y 171.806,Z 222.065,A -85,B 0,C 180,E1 -23035.307,E2 -23035.307} C_VEL
LIN {X 0,Y 172.323,Z 222.002,A -85,B 0,C 180,E1 -23040,E2 -23040} C_VEL
LIN {X 0,Y 171.817,Z 222.093,A -85,B 0,C 180,E1 -23044.692,E2 -23044.692} C_VEL
LIN {X 0,Y 172.302,Z 223.719,A -85,B 0,C 180,E1 -23049.39,E2 -23049.39} C_VEL
LIN {X 0,Y 172.526,Z 225.81,A -85,B 0,C 180,E1 -23054.147,E2 -23054.147} C_VEL
LIN {X 0,Y 173.063,Z 228.443,A -85,B 0,C 180,E1 -23058.958,E2 -23058.958} C_VEL
LIN {X 0,Y 173.754,Z 231.604,A -85,B 0,C 180,E1 -23063.859,E2 -23063.859} C_VEL
LIN {X 0,Y 174.689,Z 235.337,A -85,B 0,C 180,E1 -23068.867,E2 -23068.867} C_VEL
LIN {X 0,Y 175.811,Z 239.852,A -85,B 0,C 180,E1 -23074.031,E2 -23074.031} C_VEL
LIN {X 0,Y 176.641,Z 243.906,A -85,B 0,C 180,E1 -23078.122,E2 -23078.122} C_VEL
LIN {X 0,Y 177.817,Z 249.86,A -85,B 0,C 180,E1 -23083.511,E2 -23083.511} C_VEL
LIN {X 0,Y 179.032,Z 255.502,A -85,B 0,C 180,E1 -23088.233,E2 -23088.233} C_VEL
LIN {X 0,Y 180.022,Z 261.382,A -85,B 0,C 180,E1 -23092.767,E2 -23092.767} C_VEL
LIN {X 0,Y 179.495,Z 262.762,A -85,B 0,C 180,E1 -23093.69,E2 -23093.69} C_VEL
LIN {X 0,Y 180.571,Z 275.845,A -85,B 0,C 180,E1 -23095.086,E2 -23095.086} C_VEL
LIN {X 0,Y 180.716,Z 286.876,A -85,B 0,C 180,E1 -23096.56,E2 -23096.56} C_VEL
LIN {X 0,Y 180.246,Z 297.769,A -85,B 0,C 180,E1 -23098.374,E2 -23098.374} C_VEL
LIN {X 0,Y 179.173,Z 307.38,A -85,B 0,C 180,E1 -23100.32,E2 -23100.32} C_VEL
LIN {X 0,Y 177.936,Z 315.747,A -85,B 0,C 180,E1 -23102.352,E2 -23102.352} C_VEL
LIN {X 0,Y 176.863,Z 323.738,A -85,B 0,C 180,E1 -23104.715,E2 -23104.715} C_VEL
LIN {X 0,Y 175.257,Z 330.165,A -85,B 0,C 180,E1 -23106.911,E2 -23106.911} C_VEL
LIN {X 0,Y 173.315,Z 337.292,A -85,B 0,C 180,E1 -23109.841,E2 -23109.841} C_VEL
LIN {X 0,Y 171.685,Z 343.877,A -85,B 0,C 180,E1 -23113.352,E2 -23113.352} C_VEL
LIN {X 0,Y 170.888,Z 349.057,A -85,B 0,C 180,E1 -23116.93,E2 -23116.93} C_VEL
LIN {X 0,Y 170.824,Z 353.24,A -85,B 0,C 180,E1 -23120.897,E2 -23120.897} C_VEL
LIN {X 0,Y 171.229,Z 355.295,A -85,B 0,C 180,E1 -23123.226,E2 -23123.226} C_VEL
LIN {X 0,Y 171.267,Z 361.954,A -85,B 0,C 180,E1 -23126.474,E2 -23126.474} C_VEL
LIN {X 0,Y 171.39,Z 367.771,A -85,B 0,C 180,E1 -23130.003,E2 -23130.003} C_VEL
LIN {X 0,Y 171.049,Z 370.787,A -85,B 0,C 180,E1 -23132.358,E2 -23132.358} C_VEL
LIN {X 0,Y 170.244,Z 375.371,A -85,B 0,C 180,E1 -23137.117,E2 -23137.117} C_VEL
LIN {X 0,Y 170.468,Z 378.056,A -85,B 0,C 180,E1 -23141.085,E2 -23141.085} C_VEL
LIN {X 0,Y 170.218,Z 378.974,A -85,B 0,C 180,E1 -23143.044,E2 -23143.044} C_VEL
LIN {X 0,Y 168.587,Z 379.728,A -85,B 0,C 180,E1 -23146.342,E2 -23146.342} C_VEL
LIN {X 0,Y 167.707,Z 380.113,A -85,B 0,C 180,E1 -23149.697,E2 -23149.697} C_VEL
LIN {X 0,Y 168.614,Z 380.354,A -85,B 0,C 180,E1 -23151.677,E2 -23151.677} C_VEL
LIN {X 0,Y 173.659,Z 380.446,A -85,B 0,C 180,E1 -23156.437,E2 -23156.437} C_VEL
LIN {X 0,Y 179.504,Z 379.385,A -85,B 0,C 180,E1 -23160.599,E2 -23160.599} C_VEL
LIN {X 0,Y 186.831,Z 377.267,A -85,B 0,C 180,E1 -23164.354,E2 -23164.354} C_VEL
LIN {X 0,Y 196.241,Z 373.686,A -85,B 0,C 180,E1 -23168.011,E2 -23168.011} C_VEL
LIN {X 0,Y 207.287,Z 368.387,A -85,B 0,C 180,E1 -23171.39,E2 -23171.39} C_VEL
LIN {X 0,Y 217.781,Z 362.461,A -85,B 0,C 180,E1 -23173.937,E2 -23173.937} C_VEL
LIN {X 0,Y 228.255,Z 355.621,A -85,B 0,C 180,E1 -23176.22,E2 -23176.22} C_VEL
LIN {X 0,Y 226.783,Z 356.36,A -85,B 0,C 180,E1 -23177.017,E2 -23177.017} C_VEL
LIN {X 0,Y 216.216,Z 362.022,A -85,B 0,C 180,E1 -23179.451,E2 -23179.451} C_VEL
LIN {X 0,Y 206.235,Z 366.362,A -85,B 0,C 180,E1 -23182.164,E2 -23182.164} C_VEL
LIN {X 0,Y 195.828,Z 369.704,A -85,B 0,C 180,E1 -23185.637,E2 -23185.637} C_VEL
LIN {X 0,Y 188.711,Z 371.203,A -85,B 0,C 180,E1 -23188.575,E2 -23188.575} C_VEL
LIN {X 0,Y 181.46,Z 371.838,A -85,B 0,C 180,E1 -23192.305,E2 -23192.305} C_VEL
LIN {X 0,Y 175.356,Z 371.292,A -85,B 0,C 180,E1 -23196.373,E2 -23196.373} C_VEL
LIN {X 0,Y 170.374,Z 369.545,A -85,B 0,C 180,E1 -23200.731,E2 -23200.731} C_VEL
LIN {X 0,Y 166.55,Z 366.557,A -85,B 0,C 180,E1 -23205.334,E2 -23205.334} C_VEL
LIN {X 0,Y 164.204,Z 362.32,A -85,B 0,C 180,E1 -23210.142,E2 -23210.142} C_VEL
LIN {X 0,Y 163.063,Z 356.7,A -85,B 0,C 180,E1 -23215.055,E2 -23215.055} C_VEL
LIN {X 0,Y 162.656,Z 349.332,A -85,B 0,C 180,E1 -23220,E2 -23220} C_VEL
LIN {X 0,Y 162.798,Z 342.475,A -85,B 0,C 180,E1 -23223.713,E2 -23223.713} C_VEL
LIN {X 0,Y 163.22,Z 334.188,A -85,B 0,C 180,E1 -23227.422,E2 -23227.422} C_VEL
LIN {X 0,Y 164.017,Z 324.113,A -85,B 0,C 180,E1 -23231.118,E2 -23231.118} C_VEL
LIN {X 0,Y 165.037,Z 312.84,A -85,B 0,C 180,E1 -23234.489,E2 -23234.489} C_VEL
LIN {X 0,Y 166.241,Z 301.653,A -85,B 0,C 180,E1 -23237.214,E2 -23237.214} C_VEL
LIN {X 0,Y 167.499,Z 289.544,A -85,B 0,C 180,E1 -23239.613,E2 -23239.613} C_VEL
LIN {X 0,Y 167.598,Z 285.218,A -85,B 0,C 180,E1 -23240.341,E2 -23240.341} C_VEL
LIN {X 0,Y 165.826,Z 271.914,A -85,B 0,C 180,E1 -23242.25,E2 -23242.25} C_VEL
LIN {X 0,Y 164.554,Z 258.401,A -85,B 0,C 180,E1 -23243.77,E2 -23243.77} C_VEL
LIN {X 0,Y 165.472,Z 248.958,A -85,B 0,C 180,E1 -23249.937,E2 -23249.937} C_VEL
LIN {X 0,Y 166.505,Z 240.51,A -85,B 0,C 180,E1 -23255.477,E2 -23255.477} C_VEL
LIN {X 0,Y 166.824,Z 236.876,A -85,B 0,C 180,E1 -23257.879,E2 -23257.879} C_VEL
LIN {X 0,Y 166.359,Z 233.061,A -85,B 0,C 180,E1 -23260.494,E2 -23260.494} C_VEL
LIN {X 0,Y 165.902,Z 230.439,A -85,B 0,C 180,E1 -23262.39,E2 -23262.39} C_VEL
LIN {X 0,Y 166.351,Z 232.934,A -85,B 0,C 180,E1 -23267.467,E2 -23267.467} C_VEL
LIN {X 0,Y 166.619,Z 234.747,A -85,B 0,C 180,E1 -23270.747,E2 -23270.747} C_VEL
LIN {X 0,Y 166.931,Z 237.561,A -85,B 0,C 180,E1 -23275.362,E2 -23275.362} C_VEL
LIN {X 0,Y 166.971,Z 238.169,A -85,B 0,C 180,E1 -23276.295,E2 -23276.295} C_VEL
LIN {X 0,Y 168.48,Z 241.451,A -85,B 0,C 180,E1 -23276.98,E2 -23276.98} C_VEL
LIN {X 0,Y 171.792,Z 248.982,A -85,B 0,C 180,E1 -23278.649,E2 -23278.649} C_VEL
LIN {X 0,Y 174.535,Z 257.36,A -85,B 0,C 180,E1 -23280.554,E2 -23280.554} C_VEL
LIN {X 0,Y 176.393,Z 265.424,A -85,B 0,C 180,E1 -23282.56,E2 -23282.56} C_VEL
LIN {X 0,Y 177.36,Z 272.52,A -85,B 0,C 180,E1 -23284.48,E2 -23284.48} C_VEL
LIN {X 0,Y 177.688,Z 276.896,A -85,B 0,C 180,E1 -23285.769,E2 -23285.769} C_VEL
LIN {X 0,Y 176.014,Z 283.633,A -85,B 0,C 180,E1 -23287.705,E2 -23287.705} C_VEL
LIN {X 0,Y 173.86,Z 290.006,A -85,B 0,C 180,E1 -23289.901,E2 -23289.901} C_VEL
LIN {X 0,Y 171.297,Z 296.294,A -85,B 0,C 180,E1 -23292.692,E2 -23292.692} C_VEL
LIN {X 0,Y 169.301,Z 301.14,A -85,B 0,C 180,E1 -23295.574,E2 -23295.574} C_VEL
LIN {X 0,Y 167.867,Z 305.385,A -85,B 0,C 180,E1 -23299.138,E2 -23299.138} C_VEL
LIN {X 0,Y 166.338,Z 308.343,A -85,B 0,C 180,E1 -23302.715,E2 -23302.715} C_VEL
LIN {X 0,Y 165.849,Z 309.571,A -85,B 0,C 180,E1 -23305.135,E2 -23305.135} C_VEL
LIN {X 0,Y 165.454,Z 310.329,A -85,B 0,C 180,E1 -23307.562,E2 -23307.562} C_VEL
LIN {X 0,Y 165.307,Z 310.603,A -85,B 0,C 180,E1 -23309.997,E2 -23309.997} C_VEL
LIN {X 0,Y 165.453,Z 310.361,A -85,B 0,C 180,E1 -23312.431,E2 -23312.431} C_VEL
LIN {X 0,Y 165.847,Z 309.648,A -85,B 0,C 180,E1 -23314.859,E2 -23314.859} C_VEL
LIN {X 0,Y 166.335,Z 308.453,A -85,B 0,C 180,E1 -23317.279,E2 -23317.279} C_VEL
LIN {X 0,Y 167.852,Z 305.555,A -85,B 0,C 180,E1 -23320.857,E2 -23320.857} C_VEL
LIN {X 0,Y 169.256,Z 301.391,A -85,B 0,C 180,E1 -23324.423,E2 -23324.423} C_VEL
LIN {X 0,Y 170.242,Z 299.6,A -85,B 0,C 180,E1 -23325.562,E2 -23325.562} C_VEL
LIN {X 0,Y 171.751,Z 295.505,A -85,B 0,C 180,E1 -23327.869,E2 -23327.869} C_VEL
LIN {X 0,Y 174.366,Z 288.944,A -85,B 0,C 180,E1 -23330.648,E2 -23330.648} C_VEL
LIN {X 0,Y 177.005,Z 280.481,A -85,B 0,C 180,E1 -23333.39,E2 -23333.39} C_VEL
LIN {X 0,Y 177.781,Z 277.249,A -85,B 0,C 180,E1 -23334.276,E2 -23334.276} C_VEL
LIN {X 0,Y 176.979,Z 268.71,A -85,B 0,C 180,E1 -23336.773,E2 -23336.773} C_VEL
LIN {X 0,Y 175.198,Z 259.547,A -85,B 0,C 180,E1 -23339.092,E2 -23339.092} C_VEL
LIN {X 0,Y 172.487,Z 250.541,A -85,B 0,C 180,E1 -23341.168,E2 -23341.168} C_VEL
LIN {X 0,Y 168.663,Z 241.662,A -85,B 0,C 180,E1 -23343.145,E2 -23343.145} C_VEL
LIN {X 0,Y 167.039,Z 238.165,A -85,B 0,C 180,E1 -23343.927,E2 -23343.927} C_VEL
LIN {X 0,Y 166.899,Z 236.336,A -85,B 0,C 180,E1 -23346.862,E2 -23346.862} C_VEL
LIN {X 0,Y 166.336,Z 233.097,A -85,B 0,C 180,E1 -23352.529,E2 -23352.529} C_VEL
LIN {X 0,Y 165.973,Z 230.739,A -85,B 0,C 180,E1 -23357.35,E2 -23357.35} C_VEL
LIN {X 0,Y 165.693,Z 229.304,A -85,B 0,C 180,E1 -23360.488,E2 -23360.488} C_VEL
LIN {X 0,Y 165.406,Z 227.979,A -85,B 0,C 180,E1 -23363.827,E2 -23363.827} C_VEL
LIN {X 0,Y 165.117,Z 226.106,A -85,B 0,C 180,E1 -23369.285,E2 -23369.285} C_VEL
LIN {X 0,Y 164.833,Z 224.614,A -85,B 0,C 180,E1 -23374.762,E2 -23374.762} C_VEL
LIN {X 0,Y 164.572,Z 223.582,A -85,B 0,C 180,E1 -23380.023,E2 -23380.023} C_VEL
LIN {X 0,Y 164.533,Z 222.974,A -85,B 0,C 180,E1 -23385.782,E2 -23385.782} C_VEL
LIN {X 0,Y 164.76,Z 222.942,A -85,B 0,C 180,E1 -23390.176,E2 -23390.176} C_VEL
LIN {X 0,Y 164.763,Z 222.958,A -85,B 0,C 180,E1 -23393.878,E2 -23393.878} C_VEL
LIN {X 0,Y 165.4,Z 223.529,A -85,B 0,C 180,E1 -23400,E2 -23400} C_VEL
LIN {X 0,Y 165.253,Z 224.835,A -85,B 0,C 180,E1 -23404.879,E2 -23404.879} C_VEL
LIN {X 0,Y 165.713,Z 226.534,A -85,B 0,C 180,E1 -23409.767,E2 -23409.767} C_VEL
LIN {X 0,Y 165.957,Z 228.747,A -85,B 0,C 180,E1 -23414.72,E2 -23414.72} C_VEL
LIN {X 0,Y 166.502,Z 231.453,A -85,B 0,C 180,E1 -23419.735,E2 -23419.735} C_VEL
LIN {X 0,Y 167.236,Z 234.75,A -85,B 0,C 180,E1 -23424.85,E2 -23424.85} C_VEL
LIN {X 0,Y 168.275,Z 238.72,A -85,B 0,C 180,E1 -23430.078,E2 -23430.078} C_VEL
LIN {X 0,Y 169.026,Z 241.85,A -85,B 0,C 180,E1 -23433.744,E2 -23433.744} C_VEL
LIN {X 0,Y 169.891,Z 246.239,A -85,B 0,C 180,E1 -23438.354,E2 -23438.354} C_VEL
LIN {X 0,Y 170.843,Z 251.184,A -85,B 0,C 180,E1 -23443.039,E2 -23443.039} C_VEL
LIN {X 0,Y 172.149,Z 257.211,A -85,B 0,C 180,E1 -23448.315,E2 -23448.315} C_VEL
LIN {X 0,Y 172.993,Z 262.183,A -85,B 0,C 180,E1 -23452.271,E2 -23452.271} C_VEL
LIN {X 0,Y 173.995,Z 269.921,A -85,B 0,C 180,E1 -23453.145,E2 -23453.145} C_VEL
LIN {X 0,Y 174.494,Z 282.045,A -85,B 0,C 180,E1 -23454.702,E2 -23454.702} C_VEL
LIN {X 0,Y 174.071,Z 293.992,A -85,B 0,C 180,E1 -23456.63,E2 -23456.63} C_VEL
LIN {X 0,Y 173.023,Z 304.807,A -85,B 0,C 180,E1 -23458.786,E2 -23458.786} C_VEL
LIN {X 0,Y 171.462,Z 314.608,A -85,B 0,C 180,E1 -23461.213,E2 -23461.213} C_VEL
LIN {X 0,Y 170.22,Z 322.634,A -85,B 0,C 180,E1 -23463.654,E2 -23463.654} C_VEL
LIN {X 0,Y 169.101,Z 327.825,A -85,B 0,C 180,E1 -23465.446,E2 -23465.446} C_VEL
LIN {X 0,Y 166.536,Z 336.255,A -85,B 0,C 180,E1 -23468.983,E2 -23468.983} C_VEL
LIN {X 0,Y 164.818,Z 342.865,A -85,B 0,C 180,E1 -23472.637,E2 -23472.637} C_VEL
LIN {X 0,Y 163.867,Z 348.048,A -85,B 0,C 180,E1 -23476.36,E2 -23476.36} C_VEL
LIN {X 0,Y 163.763,Z 352.47,A -85,B 0,C 180,E1 -23480.774,E2 -23480.774} C_VEL
LIN {X 0,Y 164.371,Z 354.774,A -85,B 0,C 180,E1 -23484.021,E2 -23484.021} C_VEL
LIN {X 0,Y 164.447,Z 361.606,A -85,B 0,C 180,E1 -23487.554,E2 -23487.554} C_VEL
LIN {X 0,Y 164.562,Z 365.555,A -85,B 0,C 180,E1 -23490.003,E2 -23490.003} C_VEL
LIN {X 0,Y 164.27,Z 368.781,A -85,B 0,C 180,E1 -23492.455,E2 -23492.455} C_VEL
LIN {X 0,Y 163.406,Z 373.624,A -85,B 0,C 180,E1 -23497.417,E2 -23497.417} C_VEL
LIN {X 0,Y 163.797,Z 377.072,A -85,B 0,C 180,E1 -23502.391,E2 -23502.391} C_VEL
LIN {X 0,Y 165.502,Z 379.287,A -85,B 0,C 180,E1 -23507.296,E2 -23507.296} C_VEL
LIN {X 0,Y 168.614,Z 380.354,A -85,B 0,C 180,E1 -23511.677,E2 -23511.677} C_VEL
LIN {X 0,Y 169.757,Z 380.572,A -85,B 0,C 180,E1 -23513.641,E2 -23513.641} C_VEL
LIN {X 0,Y 170.372,Z 380.385,A -85,B 0,C 180,E1 -23516.981,E2 -23516.981} C_VEL
LIN {X 0,Y 171.701,Z 379.699,A -85,B 0,C 180,E1 -23520.26,E2 -23520.26} C_VEL
LIN {X 0,Y 173.897,Z 379.136,A -85,B 0,C 180,E1 -23522.062,E2 -23522.062} C_VEL
LIN {X 0,Y 181.035,Z 377.543,A -85,B 0,C 180,E1 -23525.617,E2 -23525.617} C_VEL
LIN {X 0,Y 189.82,Z 374.796,A -85,B 0,C 180,E1 -23529.01,E2 -23529.01} C_VEL
LIN {X 0,Y 199.533,Z 370.944,A -85,B 0,C 180,E1 -23532.01,E2 -23532.01} C_VEL
LIN {X 0,Y 210.07,Z 365.914,A -85,B 0,C 180,E1 -23534.636,E2 -23534.636} C_VEL
LIN {X 0,Y 217.063,Z 362.103,A -85,B 0,C 180,E1 -23536.129,E2 -23536.129} C_VEL
LIN {X 0,Y 217.551,Z 361.705,A -85,B 0,C 180,E1 -23536.769,E2 -23536.769} C_VEL
LIN {X 0,Y 205.898,Z 366.621,A -85,B 0,C 180,E1 -23539.569,E2 -23539.569} C_VEL
LIN {X 0,Y 195.983,Z 369.787,A -85,B 0,C 180,E1 -23542.438,E2 -23542.438} C_VEL
LIN {X 0,Y 186.926,Z 371.713,A -85,B 0,C 180,E1 -23545.669,E2 -23545.669} C_VEL
